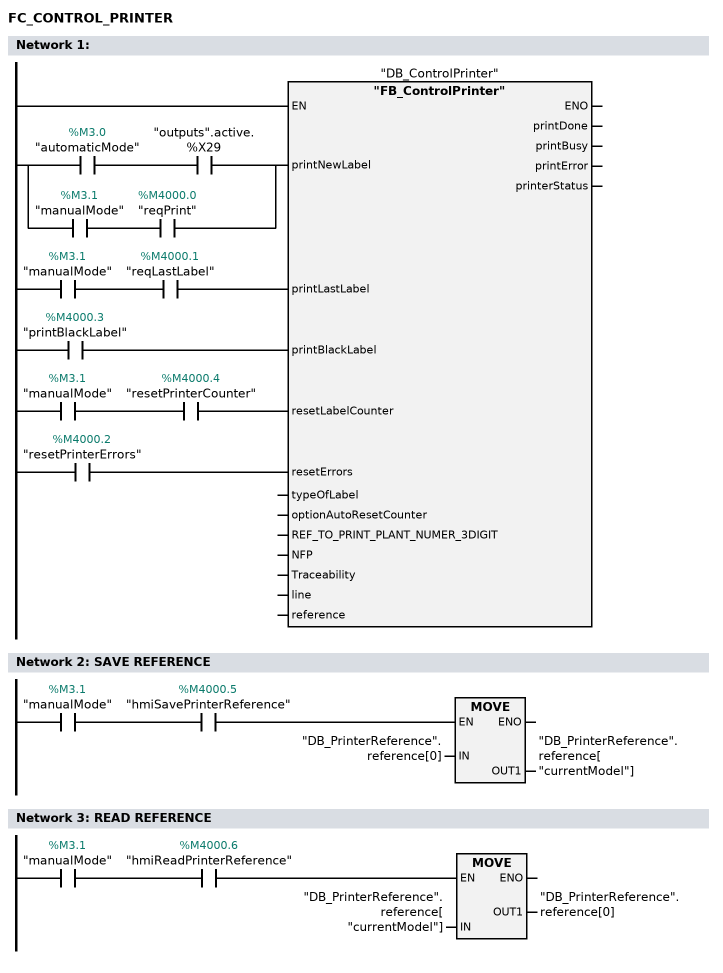
   RUNG wire#powerrail
      "DB_ControlPrinter"(printNewLabel := wire#w1, printLastLabel := wire#w2, printBlackLabel := wire#w3, resetLabelCounter := wire#w4, resetErrors := wire#w5, typeOfLabel :=, optionAutoResetCounter :=, REF_TO_PRINT_PLANT_NUMER_3DIGIT :=, NFP :=, Traceability :=, line :=, reference :=, printDone =>, printBusy =>, printError =>, printerStatus =>)
   END_RUNG
   RUNG wire#powerrail
      Contact( "automaticMode" )
      Contact( "outputs".active.%X29 )
   END_RUNG wire#w1
   RUNG wire#powerrail
      Contact( "manualMode" )
      Contact( "reqPrint" )
   END_RUNG wire#w1
   RUNG wire#powerrail
      Contact( "manualMode" )
      Contact( "reqLastLabel" )
   END_RUNG wire#w2
   RUNG wire#powerrail
      Contact( "printBlackLabel" )
   END_RUNG wire#w3
   RUNG wire#powerrail
      Contact( "manualMode" )
      Contact( "resetPrinterCounter" )
   END_RUNG wire#w4
   RUNG wire#powerrail
      Contact( "resetPrinterErrors" )
   END_RUNG wire#w5
   // the same network as SCL:
   "DB_ControlPrinter"(printNewLabel := ("automaticMode" AND "outputs".active.%X29) OR ("manualMode" AND "reqPrint"),   // "FB_ControlPrinter"
                       printLastLabel := "manualMode" AND "reqLastLabel",
                       printBlackLabel := "printBlackLabel",
                       resetLabelCounter := "manualMode" AND "resetPrinterCounter",
                       resetErrors := "resetPrinterErrors");
END_REGION

REGION Network 2: SAVE REFERENCE
   RUNG wire#powerrail
      Contact( "manualMode" )
      Contact( "hmiSavePrinterReference" )
      Move(in := "DB_PrinterReference".reference[0], out1 => "DB_PrinterReference".reference["currentModel"])
   END_RUNG
   // the same network as SCL:
   IF "manualMode" AND "hmiSavePrinterReference" THEN
       "DB_PrinterReference".reference["currentModel"] := "DB_PrinterReference".reference[0];
   END_IF;
END_REGION

REGION Network 3: READ REFERENCE
   RUNG wire#powerrail
      Contact( "manualMode" )
      Contact( "hmiReadPrinterReference" )
      Move(in := "DB_PrinterReference".reference["currentModel"], out1 => "DB_PrinterReference".reference[0])
   END_RUNG
   // the same network as SCL:
   IF "manualMode" AND "hmiReadPrinterReference" THEN
       "DB_PrinterReference".reference[0] := "DB_PrinterReference".reference["currentModel"];
   END_IF;
END_REGION
END_FUNCTION

FUNCTION_BLOCK "FB_ControlPrinter"
{ S7_Optimized_Access := 'TRUE' }
VERSION : 0.1
   VAR_INPUT 
      printNewLabel : Bool;
      printLastLabel : Bool;
      printBlackLabel : Bool;
      resetLabelCounter : Bool;
      resetErrors : Bool;
   END_VAR
   VAR_INPUT RETAIN
      typeOfLabel : Int;
   END_VAR
   VAR_INPUT 
      optionAutoResetCounter : Int;
      REF_TO_PRINT_PLANT_NUMER_3DIGIT : String[10];
      NFP : String[30];
      Traceability : Bool;
      line : String[1];
      reference : "udt_referenceMainInfo";
   END_VAR

   VAR_OUTPUT 
      printDone : Bool;
      printBusy : Bool;
      printError : Bool;
      printerStatus : Word;
   END_VAR

   VAR 
      tramToSendToPrinter : Array[0..6000] of Char;
      seqDataPreparation : Int;
      tramToPrepareToSend { S7_SetPoint := 'True'} : Array[1..20] of String;
      savePrintNewLabel : Bool;
   END_VAR
   VAR RETAIN
      "counter" : Int;
      DBcomToPrinter {InstructionName := 'TCON_IP_v4'; LibVersion := '1.0'; S7_SetPoint := 'False'} : TCON_IP_v4;
   END_VAR
   VAR 
      tSendC {InstructionName := 'TSEND_C'; LibVersion := '3.0'} : TSEND_C;
   END_VAR

   VAR_TEMP 
      dateAndTime {InstructionName := 'DTL'; LibVersion := '1.0'} : DTL;
      dateTimeStr : String;
      "date" : String[10];
      "time" : String[8];
      year : String[2];
      MFGhour : String[1];
      JulianDay : String[3];
      errCode : DInt;
      pcars : DInt;
      forCounter : Int;
      counterStr : String[4];
      cnt : DInt;
      i : Int;
      dummy : Int;
      holder : String;
      nfpToPrint : String[8];
      PN : String[8];
   END_VAR

   VAR CONSTANT 
      fieldSeparator : String := '^FS';
      RS : String := '\1E';
      GS : String := '\1D';
      EOT : String := '\04';
   END_VAR


BEGIN
	
	//***********************************************************CALCULATE DAY NUMBER **************************************
	#errCode:= RD_LOC_T(#dateAndTime);
	#dateTimeStr := "GetStrDateTime"("date" := #dateAndTime, separator := '/');
	#date := LEFT_STRING(IN := #dateTimeStr, L := 10);
	#year := MID(IN := #dateTimeStr, L := 2, P := 9);
	#time := MID(IN := #dateTimeStr, L := 8, P := 12);
	#JulianDay := "GetStrJDay"();
	#MFGhour := USINT_TO_CHAR(#dateAndTime.HOUR + 65);
	
	//********************************************* SEQUENCE MANAGE TO DATA PRINT **************************************
	//
	//>>>>>> STEP-0- >>>>>> waiting for start printing
	IF (#printNewLabel AND #seqDataPreparation = 0) THEN
	    IF #printNewLabel THEN
	        #savePrintNewLabel := TRUE;
	        #seqDataPreparation := 1;
	    END_IF;
	END_IF;
	
	//>>>>>> STEP-1- >>>>>> INITIALISE DATA TO PRINT
	IF #seqDataPreparation = 1 THEN
	    // INITILISE DATA OF TRAM TO SEND
	    // 
	    IF #typeOfLabel = 0 THEN //NO LABEL
	        FOR #i := 1 TO 20 DO
	            #tramToPrepareToSend[#i] := '';
	        END_FOR;
	        
	    ELSIF #typeOfLabel = 1 THEN //NFP LABEL
	        #tramToPrepareToSend[1] := '^XA^PW378'; //START FORMAT   
	        #tramToPrepareToSend[2] := '^BY126,126^FT169,175^BXN,7,200,0,0,1,~^FH\^FD';//DATAMATRIX
	        #tramToPrepareToSend[3] := '1234567891234567891234567891'; 
	        #tramToPrepareToSend[4] := '^FS^FT25,162^A0N,29,28^FH\^FD'; //REFERENCE
	        #tramToPrepareToSend[5] := '12345678'; 
	        #tramToPrepareToSend[6] := '^FS^FT25,124^A0N,25,24^FH\^FD'; //DATE
	        #tramToPrepareToSend[7] := 'DD/MM/YY'; //
	        #tramToPrepareToSend[8] := '^FS^FT25,87^A0N,29,28^FH\^FD'; // TIME
	        #tramToPrepareToSend[9] := 'hh:mm:ss';
	        #tramToPrepareToSend[10] := '^FS^FT26,44^A0N,29,28^FH\^FD';//DESCRIPTION
	        #tramToPrepareToSend[11] := '1234567891';
	        #tramToPrepareToSend[12] := '^FS^FT25,196^A0N,21,21^FH\^FD';//READABLE CODE
	        #tramToPrepareToSend[13] := '1234567891234567891234567891';
	        #tramToPrepareToSend[20] := '^PQ1,0,1,Y^XZ';//END FORMAT
	        #counter += 1;
	        
	    ELSIF #typeOfLabel = 2 THEN //CUSTOMER LABEL
	        #tramToPrepareToSend[1] := '^XA'; //START FORMAT   
	        #tramToPrepareToSend[2] := '^XFE:GM_FINAL.zpl';//CALL TEMPLATE
	        #tramToPrepareToSend[3] := '^FN1^FH\^FD[)>\1E06\1DY00000000000000\1DP00000000\1D12V000000000\1DT0000000000000000\1E\04^FS'; //DATAMATRIX
	        #tramToPrepareToSend[4] := '^FN2^FD1234^FS'; //GM PART NUMBER 
	        #tramToPrepareToSend[5] := '^FN3^FD5678^FS'; //GM PART NUMBER
	        #tramToPrepareToSend[6] := '^FN4^FD12345678901234^FS'; //VPPS
	        #tramToPrepareToSend[7] := '^FN5^FD123456789^FS'; //DUNS
	        #tramToPrepareToSend[8] := '^FN6^FDLSYYDDDA2B4CDSEQ^FS'; //TRACE CODE
	        #tramToPrepareToSend[9] := '^FN7^FDdd/mm/yyyy^FS'; //DATE
	        #tramToPrepareToSend[10] := '^FN8^FDhh:mm:ss^FS'; //TIME
	        #tramToPrepareToSend[11] := '^FN9^FD12345678^FS'; //FAURECIA NUMBER
	        #tramToPrepareToSend[12] := '^FN10^FD12345678^FS'; //NFP
	        #tramToPrepareToSend[13] := '^FN11^FDLINEA 3^FS'; //LINE
	        #tramToPrepareToSend[20] := '^PQ1,0,1,Y^XZ';//END FORMAT
	        #counter += 1;
	    END_IF;
	    #seqDataPreparation := 2;
	END_IF;
	
	
	//PREPARATION OF LABEL COUNTER **************************************
	#counterStr := "LabelCounterFormat"(counts := #counter, format := 'DEC', len := 3);
	IF  #counter > 999 THEN
	    #counter := 0;
	END_IF;
	
	// AUTO RESET COUNTER PER HOUR
	IF #optionAutoResetCounter = 1 THEN
	    IF #dateAndTime.MINUTE = 0 AND #dateAndTime.SECOND <= 2 THEN
	        #counter := 0;
	    END_IF;
	END_IF;
	
	
	//----------------------------------------------------------------------------------------------------------------
	//>>>>>> STEP-2- >>>>>> MODIFY CONCERNED DATA AS DATE; TIME; REFERENCE; YEAR DAY; PRODUCT REFERENCE.
	IF #seqDataPreparation = 2 THEN
	    //DATAMATRIX
	    IF #typeOfLabel = 1 THEN //NFP LABEL
	        IF #Traceability THEN
	            #tramToPrepareToSend[3] := #NFP;
	            #tramToPrepareToSend[13] := #NFP;
	        END_IF;
	        
	        IF NOT #Traceability THEN
	            #tramToPrepareToSend[3] := #line;  //line number
	            #tramToPrepareToSend[3] := CONCAT(IN1 := #tramToPrepareToSend[3], IN2 := 'P');  //label type
	            #tramToPrepareToSend[3] := CONCAT(IN1 := #tramToPrepareToSend[3], IN2 := #counterStr);  //internal sequence number
	            #tramToPrepareToSend[3] := CONCAT(IN1 := #tramToPrepareToSend[3], IN2 := #MFGhour);
	            #tramToPrepareToSend[3] := CONCAT(IN1 := #tramToPrepareToSend[3], IN2 := #JulianDay);
	            #tramToPrepareToSend[3] := CONCAT(IN1 := #tramToPrepareToSend[3], IN2 := "model".name[0]);
	            #tramToPrepareToSend[3] := CONCAT(IN1 := #tramToPrepareToSend[3], IN2 := 'R01');
	            #tramToPrepareToSend[3] := CONCAT(IN1 := #tramToPrepareToSend[3], IN2 := #REF_TO_PRINT_PLANT_NUMER_3DIGIT);
	            #tramToPrepareToSend[3] := CONCAT(IN1 := #tramToPrepareToSend[3], IN2 := #year);
	            #tramToPrepareToSend[13] := #tramToPrepareToSend[3];
	        END_IF;
	        
	        
	        //DATE
	        #tramToPrepareToSend[7] := #date;
	        
	        //TIME
	        #tramToPrepareToSend[9] := #time;
	        
	        //REFERENCE
	        #tramToPrepareToSend[5] := "model".name[0];
	        
	        //DESCRIPTION
	        #tramToPrepareToSend[11] := "model".Description[0];
	        
	        ;
	        
	        
	    ELSIF #typeOfLabel = 2 THEN //CUSTOMER LABEL
	        
	        //GM PART NUMBER 1-2
	        #tramToPrepareToSend[4] := REPLACE(IN1 := #tramToPrepareToSend[4], IN2 := (MID(IN := #reference.customerNumber, L := 4, P := 1)), L := 4, P := FIND(IN1 := #tramToPrepareToSend[4], IN2 := '1234'));
	        #tramToPrepareToSend[5] := REPLACE(IN1 := #tramToPrepareToSend[5], IN2 := (MID(IN := #reference.customerNumber, L := 4, P := 5)), L := 4, P := FIND(IN1 := #tramToPrepareToSend[5], IN2 := '5678'));
	        
	        // VPPS
	        #tramToPrepareToSend[6] := REPLACE(IN1 := #tramToPrepareToSend[6], IN2 := #reference.vpps, L := 14, P := FIND(IN1 := #tramToPrepareToSend[6], IN2 := '12345678901234'));
	        
	        // MANUFACTURING DUNS
	        #tramToPrepareToSend[7] := REPLACE(IN1 := #tramToPrepareToSend[7], IN2 := #reference.duns, L := 9, P := FIND(IN1 := #tramToPrepareToSend[7], IN2 := '123456789'));
	        
	        // TRACE CODE GM
	        //L : LINEA MACHINE
	        #tramToPrepareToSend[8] := REPLACE(IN1 := #tramToPrepareToSend[8], IN2 := #line[1], L := 1, P := (FIND(IN1 := #tramToPrepareToSend[8], IN2 := 'L')));
	        //S : SHIFT
	        #tramToPrepareToSend[8] := REPLACE(IN1 := #tramToPrepareToSend[8], IN2 := #MFGhour, L := 1, P := (FIND(IN1 := #tramToPrepareToSend[8], IN2 := 'S')));
	        //YY : YEAR
	        #tramToPrepareToSend[8] := REPLACE(IN1 := #tramToPrepareToSend[8], IN2 := #year, L := 2, P := (FIND(IN1 := #tramToPrepareToSend[8], IN2 := 'YY')));
	        //DDD : JULIAN DAY
	        #tramToPrepareToSend[8] := REPLACE(IN1 := #tramToPrepareToSend[8], IN2 := #JulianDay, L := 3, P := (FIND(IN1 := #tramToPrepareToSend[8], IN2 := 'DDD')));
	        //REF FAS 
	        #tramToPrepareToSend[8] := REPLACE(IN1 := #tramToPrepareToSend[8], IN2 := RIGHT(IN := #reference.partNumber, L := 4), L := 4, P := (FIND(IN1 := #tramToPrepareToSend[8], IN2 := 'A2B4')));
	        //REV
	        #tramToPrepareToSend[8] := REPLACE(IN1 := #tramToPrepareToSend[8], IN2 := LEFT(IN := #reference.rev, L := 2), L := 2, P := (FIND(IN1 := #tramToPrepareToSend[8], IN2 := 'CD')));
	        //SEQN : LABEL COUNTER
	        #tramToPrepareToSend[8] := REPLACE(IN1 := #tramToPrepareToSend[8], IN2 := RIGHT(IN := #counterStr, L := 3), L := 3, P := (FIND(IN1 := #tramToPrepareToSend[8], IN2 := 'SEQ')));
	        
	        
	        //Data Matrix
	        //Y : VPPS
	        #tramToPrepareToSend[3] := REPLACE(IN1 := #tramToPrepareToSend[3], IN2 := LEFT(IN := #reference.vpps, L := 14), L := 14, P := (FIND(IN1 := #tramToPrepareToSend[3], IN2 := 'Y') + 1));
	        //P : GM PART NUMBER
	        #tramToPrepareToSend[3] := REPLACE(IN1 := #tramToPrepareToSend[3], IN2 := LEFT(IN := #reference.customerNumber, L := 8), L := 8, P := (FIND(IN1 := #tramToPrepareToSend[3], IN2 := 'P') + 1));
	        //V : DUNS
	        #tramToPrepareToSend[3] := REPLACE(IN1 := #tramToPrepareToSend[3], IN2 := LEFT(IN := #reference.duns, L := 9), L := 9, P := (FIND(IN1 := #tramToPrepareToSend[3], IN2 := 'V') + 1));
	        //T : GM TRACE CODE
	        #tramToPrepareToSend[3] := REPLACE(IN1 := #tramToPrepareToSend[3], IN2 := MID(IN := #tramToPrepareToSend[8], L := 16, P := 8), L := 16, P := (FIND(IN1 := #tramToPrepareToSend[3], IN2 := 'T') + 1));
	        //DATE
	        #tramToPrepareToSend[9] := REPLACE(IN1 := #tramToPrepareToSend[9], IN2 := #date, L := 10, P := (FIND(IN1 := #tramToPrepareToSend[9], IN2 := 'dd/mm/yyyy')));
	        //TIME
	        #tramToPrepareToSend[10] := REPLACE(IN1 := #tramToPrepareToSend[10], IN2 := #time, L := 8, P := (FIND(IN1 := #tramToPrepareToSend[10], IN2 := 'hh:mm:ss')));
	        //FAURECIA NUMBER
	        #PN := MID(IN := #NFP, L := 8, P := 9);
	        #tramToPrepareToSend[11] := REPLACE(IN1 := #tramToPrepareToSend[11], IN2 := #PN, L := 8, P := (FIND(IN1 := #tramToPrepareToSend[11], IN2 := '12345678')));
	        //NFP
	        #nfpToPrint := LEFT(IN := #NFP, L := 8);
	        #tramToPrepareToSend[12] := REPLACE(IN1 := #tramToPrepareToSend[12], IN2 := #nfpToPrint, L := 8, P := (FIND(IN1 := #tramToPrepareToSend[12], IN2 := '12345678')));
	    END_IF;
	    #seqDataPreparation := 3;
	END_IF;
	
	
	//>>>>>> STEP-3- >>>>>> COPY TO TRAM PRINTER TO SEND
	IF #seqDataPreparation = 3 THEN
	    //RESET DB TRAM TO SEND 
	    FILL_BLK(IN := ' ',
	             COUNT := 6000,
	             OUT => #tramToSendToPrinter[0]);
	    #pcars := 0;
	   // FILL TRAM TO SEND TO PRINTER
	    FOR #forCounter := 1 TO 20 DO
	        Strg_TO_Chars(Strg := #tramToPrepareToSend[#forCounter],
	                      pChars := #pcars,
	                      Cnt => #cnt,
	                      Chars := #tramToSendToPrinter);
	        #pcars := #pcars + #cnt;
	    END_FOR;
	    #seqDataPreparation := 4;
	END_IF;
	
	// CONNECTION TO PRINTER PARAMETERS
	#DBcomToPrinter.ConnectionType := 16#0B;
	#DBcomToPrinter.InterfaceId := 64;
	#DBcomToPrinter.ID := 10;
	#DBcomToPrinter.ActiveEstablished := TRUE;
	#DBcomToPrinter.LocalPort := 0;
	#tSendC(REQ:=(#seqDataPreparation = 4),
	        CONT:=TRUE,
	        LEN:=0,
	        DONE=>#printDone,
	        BUSY=>#printBusy,
	        ERROR=>#printError,
	        STATUS=>#printerStatus,
	        CONNECT:=#DBcomToPrinter,
	        DATA:=#tramToSendToPrinter
	);
	IF #seqDataPreparation = 4 AND #printNewLabel THEN
	    #printDone := TRUE;
	    ;
	END_IF;
	
	
	//>>>>>> STEP-X- >>>>>> END OF SEQUENCE: WAITING 
	//
	IF #seqDataPreparation = 4 AND NOT (#printNewLabel) THEN
	    #printDone := FALSE;
	    #savePrintNewLabel := FALSE;
	    #seqDataPreparation := 0;
	END_IF;
	
	
END_FUNCTION_BLOCK

FUNCTION "GetStrJDay" : String
{ S7_Optimized_Access := 'TRUE' }
VERSION : 0.1
   VAR_TEMP 
      julianDayDint : DInt;
      DateTime {InstructionName := 'DTL'; LibVersion := '1.0'} : DTL;
      return : Int;
      LeapYear : DInt;
      julianDayHolder : String;
   END_VAR

   VAR CONSTANT 
      "__JAN" : USInt := 1;
      "__FEB" : USInt := 2;
      "__MAR" : USInt := 3;
      "__APR" : USInt := 4;
      "__MAY" : USInt := 5;
      "__JUN" : USInt := 6;
      "__JUL" : USInt := 7;
      "__AUG" : USInt := 8;
      "__SEP" : USInt := 9;
      "__OCT" : USInt := 10;
      "__NOV" : USInt := 11;
      "__DEC" : USInt := 12;
   END_VAR


BEGIN
	#return := RD_LOC_T(#DateTime);
	#LeapYear := #DateTime.YEAR MOD 4;
	
	//CALC JDAY
	CASE #DateTime.MONTH OF
	    #"__JAN": #julianDayDint := #DateTime.DAY;
	    #"__FEB": #julianDayDint := (#DateTime.DAY + DINT#31);
	    #"__MAR": #julianDayDint := (#DateTime.DAY + DINT#59);
	    #"__APR": #julianDayDint := (#DateTime.DAY + DINT#90);
	    #"__MAY": #julianDayDint := (#DateTime.DAY + DINT#120);
	    #"__JUN": #julianDayDint := (#DateTime.DAY + DINT#151);
	    #"__JUL": #julianDayDint := (#DateTime.DAY + DINT#181);
	    #"__AUG": #julianDayDint := (#DateTime.DAY + DINT#212);
	    #"__SEP": #julianDayDint := (#DateTime.DAY + DINT#243);
	    #"__OCT": #julianDayDint := (#DateTime.DAY + DINT#273);
	    #"__NOV": #julianDayDint := (#DateTime.DAY + DINT#304);
	    #"__DEC": #julianDayDint := (#DateTime.DAY + DINT#334);
	END_CASE;
	
	//IF LEAP YEAR
	IF #LeapYear = 0 AND #DateTime.MONTH > 2 THEN
	    #julianDayDint := #julianDayDint + 1;
	    ;
	END_IF;
	
	//JULIAN DAY IN STRING FORMAT
	#julianDayHolder := DINT_TO_STRING(IN := ABS_DINT(IN := #julianDayDint));
	#julianDayHolder := DELETE(IN := #julianDayHolder, L := 1, P := 1);
	IF #julianDayDint < 10 THEN
	    #GetStrJDay := CONCAT_STRING(IN1 := '00', IN2 := #julianDayHolder);
	ELSIF #julianDayDint >= 10 AND #julianDayDint < 100 THEN
	    #GetStrJDay := CONCAT_STRING(IN1 := '0', IN2 := #julianDayHolder);
	ELSE
	    #GetStrJDay := #julianDayHolder;
	END_IF;
	
	
END_FUNCTION

FUNCTION "LabelCounterFormat" : String
{ S7_Optimized_Access := 'TRUE' }
VERSION : 0.1
   VAR_INPUT 
      counts : Int;
      format : String;
      len : Int;
   END_VAR

   VAR_TEMP 
      tempCounter : String;
      i : Int;
      errCode : Word;
   END_VAR


BEGIN
	
	IF #format = 'DEC' THEN
	    VAL_STRG(IN := #counts,
	             SIZE := INT_TO_USINT( #len),
	             PREC := 0,
	             FORMAT := 0,
	             P := 1,
	             OUT => #tempCounter);
	    FOR #i := 0 TO #len DO
	        IF (FIND(IN1 := #tempCounter, IN2 := ' ') > 0) THEN
	            #tempCounter := REPLACE(IN1 := #tempCounter, IN2 := '0', L := 1, P := FIND(IN1 := #tempCounter, IN2 := ' '));
	        END_IF;
	    END_FOR;
	ELSIF #format = 'HEX' THEN
	    #errCode := HTA(IN := #counts, N := INT_TO_USINT(#len), OUT => #tempCounter);
	
	END_IF;
	#LabelCounterFormat := #tempCounter;
END_FUNCTION

FUNCTION_BLOCK "FC_IJCORE_MAIN"   // FB1000, LAD
{ S7_Optimized_Access := 'FALSE' }
VERSION : 0.1
// stored: AutoNumber false, IsIECCheckEnabled false, SetENOAutomatically false, UDAEnableTagReadback false
   VAR DB_SPECIFIC
      Enable : Bool;
      Mode : Int;
      Indicator : Int;
      AlarmReset : Bool;
      NFP : Array[1..5] of String[30];
   END_VAR
   VAR
      AWK : "FB_IJC_AWAKE_SIGNAL";
      MSG : Array[1..20] of "FB_IJC_PROTOCOL";
   END_VAR
   VAR DB_SPECIFIC
      Faults : Array[0..1] of Word;
   END_VAR
   VAR
      FaultsArray AT Faults : Array[1..32] of Bool;
   END_VAR
   VAR_TEMP
      "return" : Bool;
      i : Int;
      ERROR_STR : String;
   END_VAR
BEGIN

REGION Network 1: Fault Reset
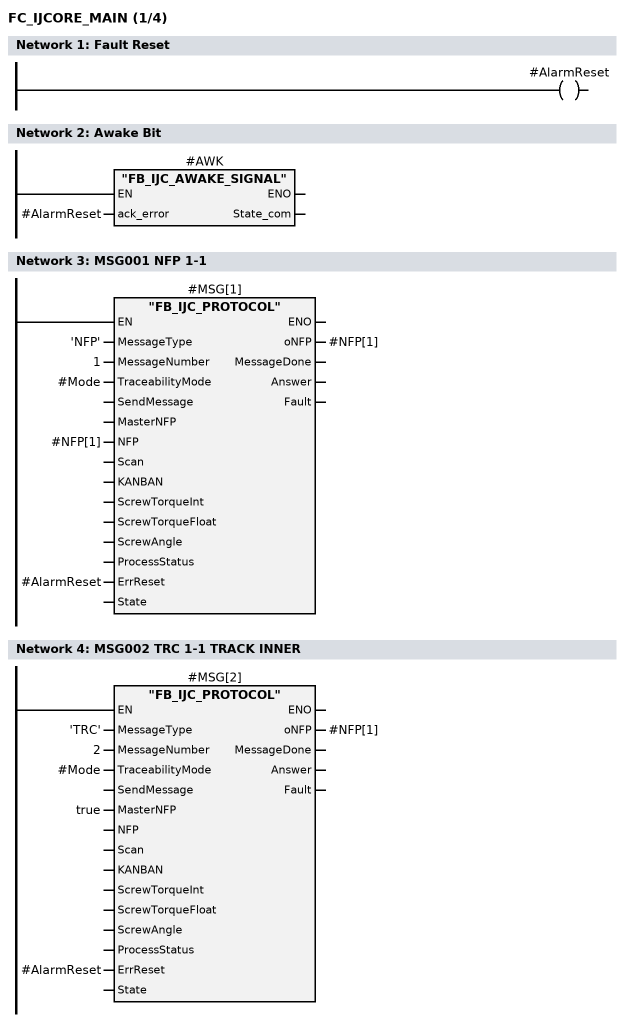
   RUNG wire#powerrail
      Coil( #AlarmReset )
   END_RUNG
   // the same network as SCL:
   #AlarmReset := TRUE;
END_REGION

REGION Network 2: Awake Bit
   RUNG wire#powerrail
      #AWK(ack_error := #AlarmReset, State_com =>)
   END_RUNG
   // the same network as SCL:
   #AWK(ack_error := #AlarmReset);   // "FB_IJC_AWAKE_SIGNAL"
END_REGION

REGION Network 3: MSG001 NFP 1-1
   RUNG wire#powerrail
      #MSG[1](MessageType := 'NFP', MessageNumber := 1, TraceabilityMode := #Mode, SendMessage :=, MasterNFP :=, NFP := #NFP[1], Scan :=, KANBAN :=, ScrewTorqueInt :=, ScrewTorqueFloat :=, ScrewAngle :=, ProcessStatus :=, ErrReset := #AlarmReset, State :=, oNFP => #NFP[1], MessageDone =>, Answer =>, Fault =>)
   END_RUNG
   // the same network as SCL:
   #MSG[1](MessageType := 'NFP',   // "FB_IJC_PROTOCOL"
           MessageNumber := 1,
           TraceabilityMode := #Mode,
           NFP := #NFP[1],
           ErrReset := #AlarmReset,
           oNFP => #NFP[1]);
END_REGION

REGION Network 4: MSG002 TRC 1-1 TRACK INNER
   RUNG wire#powerrail
      #MSG[2](MessageType := 'TRC', MessageNumber := 2, TraceabilityMode := #Mode, SendMessage :=, MasterNFP := true, NFP :=, Scan :=, KANBAN :=, ScrewTorqueInt :=, ScrewTorqueFloat :=, ScrewAngle :=, ProcessStatus :=, ErrReset := #AlarmReset, State :=, oNFP => #NFP[1], MessageDone =>, Answer =>, Fault =>)
   END_RUNG
   // the same network as SCL:
   #MSG[2](MessageType := 'TRC',   // "FB_IJC_PROTOCOL"
           MessageNumber := 2,
           TraceabilityMode := #Mode,
           MasterNFP := true,
           ErrReset := #AlarmReset,
           oNFP => #NFP[1]);
END_REGION

REGION Network 5: MSG003 TRC 1-2 TRACK OUTER
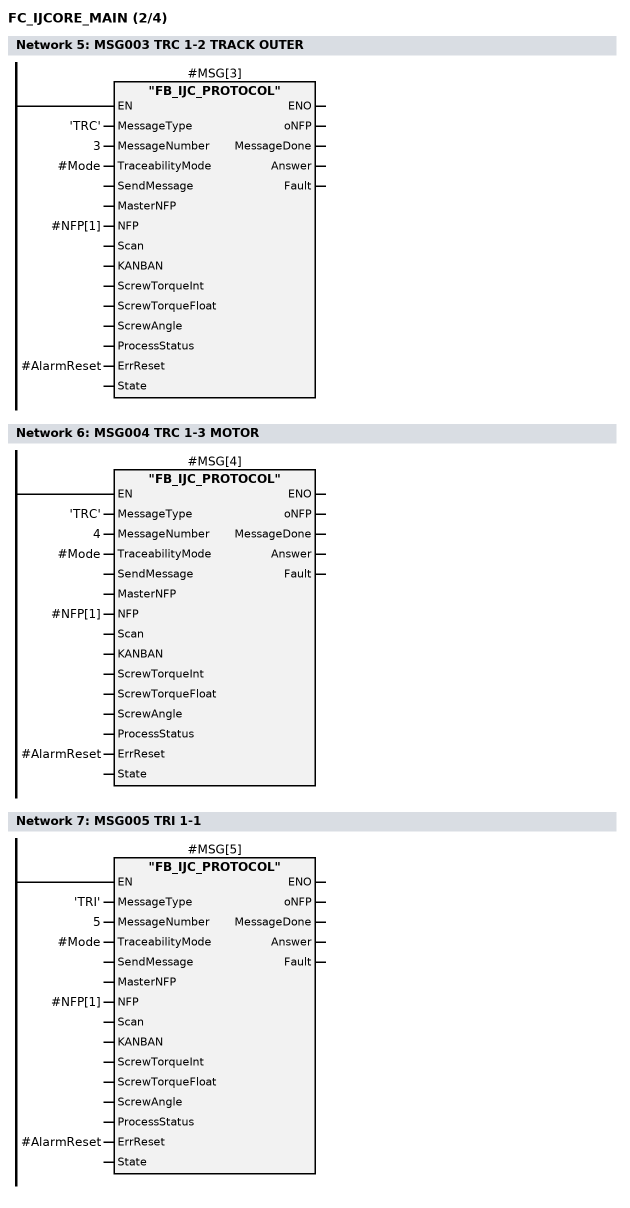
   RUNG wire#powerrail
      #MSG[3](MessageType := 'TRC', MessageNumber := 3, TraceabilityMode := #Mode, SendMessage :=, MasterNFP :=, NFP := #NFP[1], Scan :=, KANBAN :=, ScrewTorqueInt :=, ScrewTorqueFloat :=, ScrewAngle :=, ProcessStatus :=, ErrReset := #AlarmReset, State :=, oNFP =>, MessageDone =>, Answer =>, Fault =>)
   END_RUNG
   // the same network as SCL:
   #MSG[3](MessageType := 'TRC',   // "FB_IJC_PROTOCOL"
           MessageNumber := 3,
           TraceabilityMode := #Mode,
           NFP := #NFP[1],
           ErrReset := #AlarmReset);
END_REGION

REGION Network 6: MSG004 TRC 1-3 MOTOR
   RUNG wire#powerrail
      #MSG[4](MessageType := 'TRC', MessageNumber := 4, TraceabilityMode := #Mode, SendMessage :=, MasterNFP :=, NFP := #NFP[1], Scan :=, KANBAN :=, ScrewTorqueInt :=, ScrewTorqueFloat :=, ScrewAngle :=, ProcessStatus :=, ErrReset := #AlarmReset, State :=, oNFP =>, MessageDone =>, Answer =>, Fault =>)
   END_RUNG
   // the same network as SCL:
   #MSG[4](MessageType := 'TRC',   // "FB_IJC_PROTOCOL"
           MessageNumber := 4,
           TraceabilityMode := #Mode,
           NFP := #NFP[1],
           ErrReset := #AlarmReset);
END_REGION

REGION Network 7: MSG005 TRI 1-1
   RUNG wire#powerrail
      #MSG[5](MessageType := 'TRI', MessageNumber := 5, TraceabilityMode := #Mode, SendMessage :=, MasterNFP :=, NFP := #NFP[1], Scan :=, KANBAN :=, ScrewTorqueInt :=, ScrewTorqueFloat :=, ScrewAngle :=, ProcessStatus :=, ErrReset := #AlarmReset, State :=, oNFP =>, MessageDone =>, Answer =>, Fault =>)
   END_RUNG
   // the same network as SCL:
   #MSG[5](MessageType := 'TRI',   // "FB_IJC_PROTOCOL"
           MessageNumber := 5,
           TraceabilityMode := #Mode,
           NFP := #NFP[1],
           ErrReset := #AlarmReset);
END_REGION

REGION Network 8: MSG006 CNF 1-1 TRACK INNER
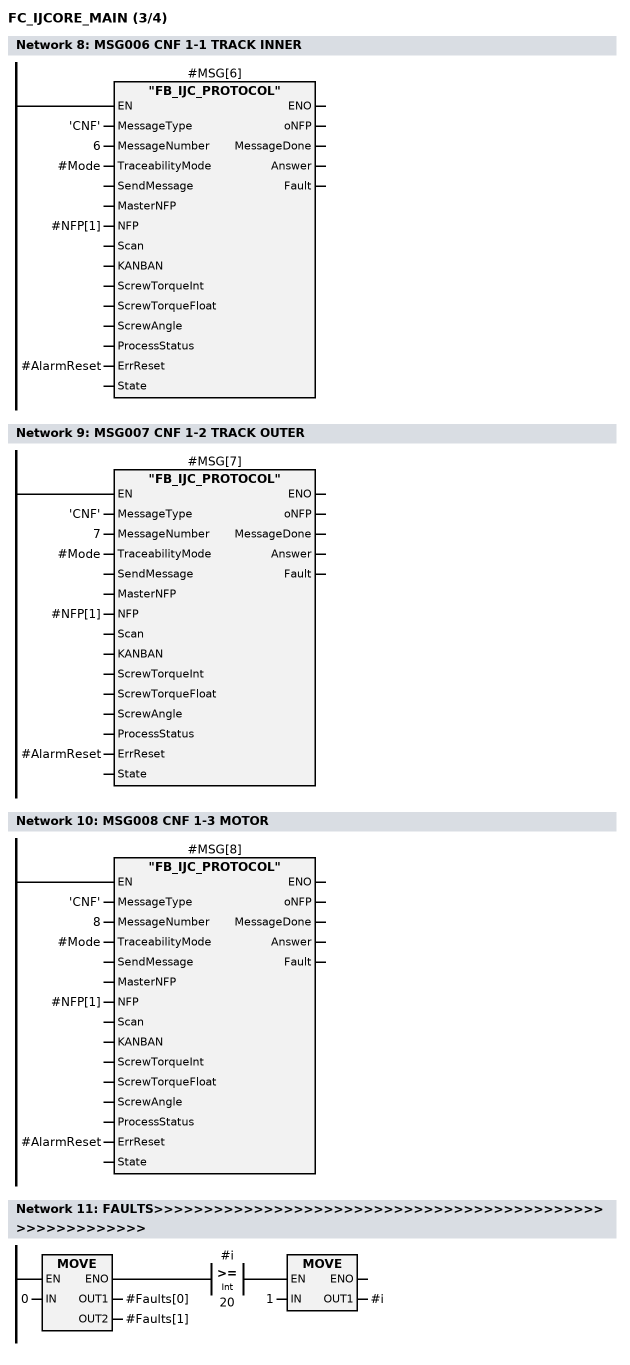
   RUNG wire#powerrail
      #MSG[6](MessageType := 'CNF', MessageNumber := 6, TraceabilityMode := #Mode, SendMessage :=, MasterNFP :=, NFP := #NFP[1], Scan :=, KANBAN :=, ScrewTorqueInt :=, ScrewTorqueFloat :=, ScrewAngle :=, ProcessStatus :=, ErrReset := #AlarmReset, State :=, oNFP =>, MessageDone =>, Answer =>, Fault =>)
   END_RUNG
   // the same network as SCL:
   #MSG[6](MessageType := 'CNF',   // "FB_IJC_PROTOCOL"
           MessageNumber := 6,
           TraceabilityMode := #Mode,
           NFP := #NFP[1],
           ErrReset := #AlarmReset);
END_REGION

REGION Network 9: MSG007 CNF 1-2 TRACK OUTER
   RUNG wire#powerrail
      #MSG[7](MessageType := 'CNF', MessageNumber := 7, TraceabilityMode := #Mode, SendMessage :=, MasterNFP :=, NFP := #NFP[1], Scan :=, KANBAN :=, ScrewTorqueInt :=, ScrewTorqueFloat :=, ScrewAngle :=, ProcessStatus :=, ErrReset := #AlarmReset, State :=, oNFP =>, MessageDone =>, Answer =>, Fault =>)
   END_RUNG
   // the same network as SCL:
   #MSG[7](MessageType := 'CNF',   // "FB_IJC_PROTOCOL"
           MessageNumber := 7,
           TraceabilityMode := #Mode,
           NFP := #NFP[1],
           ErrReset := #AlarmReset);
END_REGION

REGION Network 10: MSG008 CNF 1-3 MOTOR
   RUNG wire#powerrail
      #MSG[8](MessageType := 'CNF', MessageNumber := 8, TraceabilityMode := #Mode, SendMessage :=, MasterNFP :=, NFP := #NFP[1], Scan :=, KANBAN :=, ScrewTorqueInt :=, ScrewTorqueFloat :=, ScrewAngle :=, ProcessStatus :=, ErrReset := #AlarmReset, State :=, oNFP =>, MessageDone =>, Answer =>, Fault =>)
   END_RUNG
   // the same network as SCL:
   #MSG[8](MessageType := 'CNF',   // "FB_IJC_PROTOCOL"
           MessageNumber := 8,
           TraceabilityMode := #Mode,
           NFP := #NFP[1],
           ErrReset := #AlarmReset);
END_REGION

REGION Network 11: FAULTS>>>>>>>>>>>>>>>>>>>>>>>>>>>>>>>>>>>>>>>>>>>>>>>>>>>>>>>>>>
   RUNG wire#powerrail
      Move(in := 0, out1 => #Faults[0], out2 => #Faults[1])
      { S7_Templates := "SrcType := Int" } GE_Contact(in1 := #i, in2 := 20)
      Move(in := 1, out1 => #i)
   END_RUNG
   // the same network as SCL:
   #Faults[0] := 0;
   #Faults[1] := 0;
   IF #i >= 20 THEN #i := 1; END_IF;
END_REGION

REGION Network 12: Awake bit
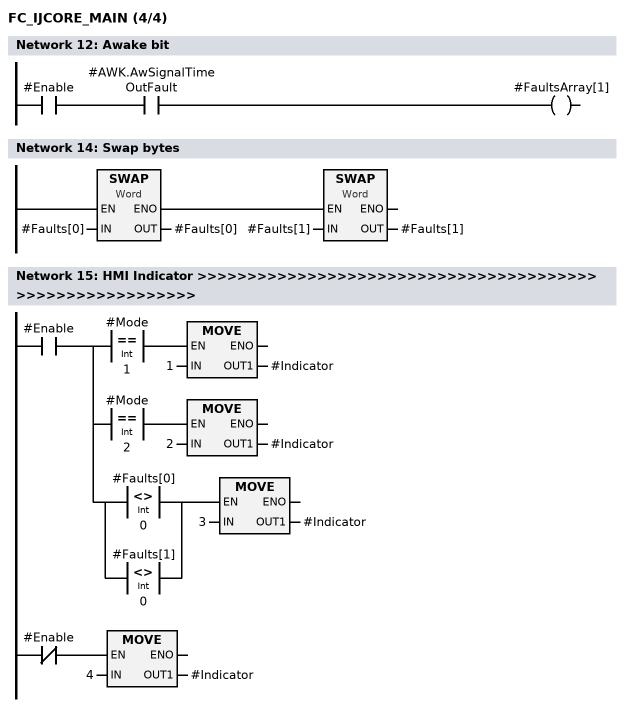
   RUNG wire#powerrail
      Contact( #Enable )
      Contact( #AWK.AwSignalTimeOutFault )
      Coil( #FaultsArray[1] )
   END_RUNG
   // the same network as SCL:
   #FaultsArray[1] := #Enable AND #AWK.AwSignalTimeOutFault;
END_REGION

REGION Network 13 (SCL): Answer faults
   FOR #i := 1 TO 20 DO
       CASE #MSG[#i].Answer OF
           -2:  // NFP not founded
               #FaultsArray[2] := TRUE;
           -3:  //Part number NOT inside BOM
               #FaultsArray[3] := TRUE;
           -4: // PFC not ok
               #FaultsArray[4] := TRUE;
           -5: //Component already used
               #FaultsArray[5] := true;
           -6: //Module already used
               #FaultsArray[6] := true;
           -10: //Status NOK from previous operation
               #FaultsArray[10] := true;

       END_CASE;



   END_FOR;
END_REGION

REGION Network 14: Swap bytes
   #Faults[0] := SWAP(#Faults[0]);
   #Faults[1] := SWAP(#Faults[1]);
END_REGION

REGION Network 15: HMI Indicator >>>>>>>>>>>>>>>>>>>>>>>>>>>>>>>>>>>>>>>>>>>>>>>>>>>>>>>>>>
   RUNG wire#powerrail
      Contact( #Enable )
      wire#w1
      { S7_Templates := "SrcType := Int" } EQ_Contact(in1 := #Mode, in2 := 1)
      Move(in := 1, out1 => #Indicator)
   END_RUNG
   RUNG wire#w1
      { S7_Templates := "SrcType := Int" } EQ_Contact(in1 := #Mode, in2 := 2)
      Move(in := 2, out1 => #Indicator)
   END_RUNG
   RUNG wire#w1
      { S7_Templates := "SrcType := Int" } NE_Contact(in1 := #Faults[0], in2 := 0)
      wire#w2
      Move(in := 3, out1 => #Indicator)
   END_RUNG
   RUNG wire#w1
      { S7_Templates := "SrcType := Int" } NE_Contact(in1 := #Faults[1], in2 := 0)
   END_RUNG wire#w2
   RUNG wire#powerrail
      I_Contact( #Enable )
      Move(in := 4, out1 => #Indicator)
   END_RUNG
   // the same network as SCL:
   IF #Enable AND (#Mode = 1) THEN #Indicator := 1; END_IF;
   IF #Enable AND (#Mode = 2) THEN #Indicator := 2; END_IF;
   IF #Enable AND ((#Faults[0] <> 0) OR (#Faults[1] <> 0)) THEN #Indicator := 3; END_IF;
   IF NOT #Enable THEN #Indicator := 4; END_IF;
END_REGION
END_FUNCTION_BLOCK

FUNCTION_BLOCK "FB_IJC_AWAKE_SIGNAL"   // FB1003, LAD
TITLE = Awake signal
{ S7_Optimized_Access := 'TRUE' }
VERSION : 0.1
// This function supervise Awake signal, 
// - Awake signal is to test communication between PLC and IJCORE. 
// - Awake signal is set to 1 by PLC and set to -1 by IJCORE alternatively.
// - first PLC check if awake signal is different of 1, if it is, PLC launch timer T1 
//  (1s<T1<10s). at the end of this temporisation, PLC set awake signal to 1 and 
//  launch Timer 2. 
// - if IJCORE don't set awake signal to -1 before the end of timer 2,PLC generate  
//   Time out fault for awake signal.
// stored: AutoNumber false, IsIECCheckEnabled false, IsRetainMemResEnabled false, MemoryReserve 100, SetENOAutomatically false, UDAEnableTagReadback false
   VAR_INPUT
      ack_error : Bool;
   END_VAR
   VAR_OUTPUT
      State_com : SInt;
   END_VAR
   VAR
      T1PresetValue : Time := T#1S;
      T2PresetValue : Time := T#60S;
      AwSignalTimeOutFault : Bool := 0;
      Reset_Counters : Bool;
      Restart_Counter_bit_of_life : USInt := 0;
      NB_Bit_of_Life : Bool;
      number_restart : DInt;
      check_restart : Bool;
      "Timer" { ExternalAccessible := 'False'; ExternalVisible := 'False'; ExternalWritable := 'False'} : Array[1..5] of TON_TIME;
   END_VAR
   VAR CONSTANT
      Trestart : Time := T#200ms;
      T3 : Time := T#2s;
   END_VAR
   VAR_TEMP   // added for the SCL form of the ladder/FBD networks
      _w1 : Bool;
   END_VAR
BEGIN

REGION Network 1: - if awake signal is -1 then launch timer 1
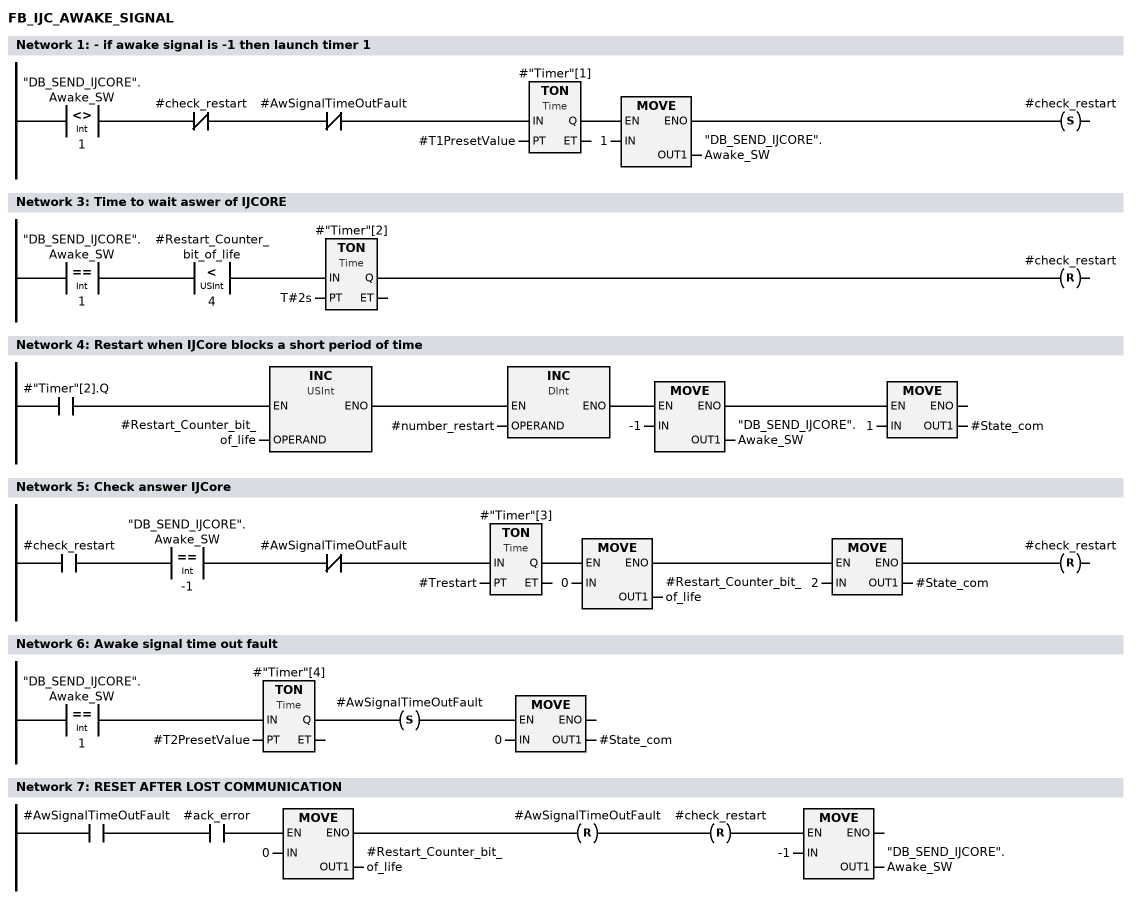
   RUNG wire#powerrail
      { S7_Templates := "SrcType := Int" } NE_Contact(in1 := "DB_SEND_IJCORE".Awake_SW, in2 := 1)
      I_Contact( #check_restart )
      I_Contact( #AwSignalTimeOutFault )
      { S7_Templates := "time_type := Time" } #"Timer"[1].TON(pt := #T1PresetValue, et =>)
      Move(in := 1, out1 => "DB_SEND_IJCORE".Awake_SW)
      S_Coil( #check_restart )
   END_RUNG
   // the same network as SCL:
   #"Timer"[1].TON(IN := ("DB_SEND_IJCORE".Awake_SW <> 1) AND NOT #check_restart AND NOT #AwSignalTimeOutFault,
                   PT := #T1PresetValue);
   IF #"Timer"[1].Q THEN
       "DB_SEND_IJCORE".Awake_SW := 1;
       #check_restart := TRUE;
   END_IF;
END_REGION

REGION Network 2: Diagnostic
END_REGION

REGION Network 3: Time to wait aswer of IJCORE
   RUNG wire#powerrail
      { S7_Templates := "SrcType := Int" } EQ_Contact(in1 := "DB_SEND_IJCORE".Awake_SW, in2 := 1)
      { S7_Templates := "SrcType := USInt" } LT_Contact(in1 := #Restart_Counter_bit_of_life, in2 := 4)
      { S7_Templates := "time_type := Time" } #"Timer"[2].TON(pt := T#2s, et =>)
      R_Coil( #check_restart )
   END_RUNG
   // the same network as SCL:
   #"Timer"[2].TON(IN := ("DB_SEND_IJCORE".Awake_SW = 1) AND (#Restart_Counter_bit_of_life < 4), PT := T#2s);
   IF #"Timer"[2].Q THEN #check_restart := FALSE; END_IF;
END_REGION

REGION Network 4: Restart when IJCore blocks a short period of time
   RUNG wire#powerrail
      Contact( #"Timer"[2].Q )
      { S7_Templates := "DestType := USInt" } Inc( #Restart_Counter_bit_of_life )
      { S7_Templates := "DestType := DInt" } Inc( #number_restart )
      Move(in := -1, out1 => "DB_SEND_IJCORE".Awake_SW)
      Move(in := 1, out1 => #State_com)
   END_RUNG
   // the same network as SCL:
   IF #"Timer"[2].Q THEN
       #Restart_Counter_bit_of_life := #Restart_Counter_bit_of_life + 1;
       #number_restart := #number_restart + 1;
       "DB_SEND_IJCORE".Awake_SW := -1;
       #State_com := 1;
   END_IF;
END_REGION

REGION Network 5: Check answer IJCore
   RUNG wire#powerrail
      Contact( #check_restart )
      { S7_Templates := "SrcType := Int" } EQ_Contact(in1 := "DB_SEND_IJCORE".Awake_SW, in2 := -1)
      I_Contact( #AwSignalTimeOutFault )
      { S7_Templates := "time_type := Time" } #"Timer"[3].TON(pt := #Trestart, et =>)
      Move(in := 0, out1 => #Restart_Counter_bit_of_life)
      Move(in := 2, out1 => #State_com)
      R_Coil( #check_restart )
   END_RUNG
   // the same network as SCL:
   #"Timer"[3].TON(IN := #check_restart AND ("DB_SEND_IJCORE".Awake_SW = (-1)) AND NOT #AwSignalTimeOutFault,
                   PT := #Trestart);
   IF #"Timer"[3].Q THEN
       #Restart_Counter_bit_of_life := 0;
       #State_com := 2;
       #check_restart := FALSE;
   END_IF;
END_REGION

REGION Network 6: Awake signal time out fault
   RUNG wire#powerrail
      { S7_Templates := "SrcType := Int" } EQ_Contact(in1 := "DB_SEND_IJCORE".Awake_SW, in2 := 1)
      { S7_Templates := "time_type := Time" } #"Timer"[4].TON(pt := #T2PresetValue, et =>)
      S_Coil( #AwSignalTimeOutFault )
      Move(in := 0, out1 => #State_com)
   END_RUNG
   // the same network as SCL:
   #"Timer"[4].TON(IN := "DB_SEND_IJCORE".Awake_SW = 1, PT := #T2PresetValue);
   IF #"Timer"[4].Q THEN
       #AwSignalTimeOutFault := TRUE;
       #State_com := 0;
   END_IF;
END_REGION

REGION Network 7: RESET AFTER LOST COMMUNICATION
   RUNG wire#powerrail
      Contact( #AwSignalTimeOutFault )
      Contact( #ack_error )
      Move(in := 0, out1 => #Restart_Counter_bit_of_life)
      R_Coil( #AwSignalTimeOutFault )
      R_Coil( #check_restart )
      Move(in := -1, out1 => "DB_SEND_IJCORE".Awake_SW)
   END_RUNG
   // the same network as SCL:
   IF #AwSignalTimeOutFault AND #ack_error THEN #Restart_Counter_bit_of_life := 0; END_IF;
   #_w1 := #AwSignalTimeOutFault AND #ack_error;
   IF #_w1 THEN
       #AwSignalTimeOutFault := FALSE;
       #check_restart := FALSE;
       "DB_SEND_IJCORE".Awake_SW := -1;
   END_IF;
END_REGION
END_FUNCTION_BLOCK

FUNCTION_BLOCK "FB_IJC_PROTOCOL"
TITLE = IJCORE PROTOCOL
{ S7_Optimized_Access := 'TRUE' }
AUTHOR : 'R.ROBINS'
VERSION : 0.1
   VAR_INPUT 
      MessageType : String[3];
      MessageNumber { ExternalVisible := 'False'; ExternalWritable := 'False'} : DInt;
      TraceabilityMode : Int;
      SendMessage { ExternalVisible := 'False'; ExternalWritable := 'False'} : Bool;
      MasterNFP : Bool;
      NFP : String[30];
      Scan : String[80];
      KANBAN : String[11];
      ScrewTorqueInt : Word;
      ScrewTorqueFloat : Word;
      ScrewAngle : Word;
      ProcessStatus { ExternalAccessible := 'False'; ExternalVisible := 'False'; ExternalWritable := 'False'} : USInt;
      ErrReset { ExternalAccessible := 'False'; ExternalVisible := 'False'; ExternalWritable := 'False'} : Bool;
   END_VAR

   VAR_OUTPUT 
      oNFP : String[30];
      MessageDone : Bool;
      Answer : Int;
      Fault : DInt;
   END_VAR

   VAR_IN_OUT 
      State { ExternalAccessible := 'False'; ExternalVisible := 'False'; ExternalWritable := 'False'} : Int;
   END_VAR

   VAR 
      SEND_OFFSET { ExternalAccessible := 'False'; ExternalVisible := 'False'; ExternalWritable := 'False'} : Struct
         SW { ExternalAccessible := 'False'; ExternalVisible := 'False'; ExternalWritable := 'False'} : DInt;
         MSG { ExternalAccessible := 'False'; ExternalVisible := 'False'; ExternalWritable := 'False'} : DInt;
      END_STRUCT;
      REC_OFFSET { ExternalAccessible := 'False'; ExternalVisible := 'False'; ExternalWritable := 'False'} : Struct
         SW { ExternalAccessible := 'False'; ExternalVisible := 'False'; ExternalWritable := 'False'} : DInt;
         MSG { ExternalAccessible := 'False'; ExternalVisible := 'False'; ExternalWritable := 'False'} : DInt;
         ANS { ExternalAccessible := 'False'; ExternalVisible := 'False'; ExternalWritable := 'False'} : DInt;
      END_STRUCT;
      ONS : Array[1..8] of Bool;
   END_VAR

   VAR_TEMP 
      IDB : Int;
      i : Int;
      j : Int;
      k : Int;
      CNT : Int;
      CNT_STR : String[2];
      MSG : DInt;
      ErrCode : Int;
   END_VAR

   VAR CONSTANT 
      "DB" : Byte := 16#84;
      CLEAR : Word := 16#0000;
      MINUS1 : Word := 16#FFFF;
      PLUS1 : Word := 16#0001;
      DB_REC : DB_ANY := 1006;
      DB_SEND : DB_ANY := 1005;
      "_CNF_" : Int := 1;
      "_TRS_" : Int := 2;
      "_TRI_" : Int := 3;
      "_TRE_" : Int := 4;
      "_STA_" : Int := 5;
      "_ANDON_" : Int := 6;
      "_TRR_" : Int := 7;
      "_TRW_" : Int := 8;
      "_PFC_" : Int := 9;
      "_NFP_" : Int := 10;
      "_CMA_" : Int := 11;
      "_TMA_" : Int := 12;
      "_TRB_" : Int := 13;
      Blank : String := '';
   END_VAR


BEGIN
	//TITLE = 'IJCORE PROTOCOL'
	//AUTHOR: RAUL ROBINS
	//CREATED ON: 03/24/2023
	//VERSION: 3.0
	
	
	
	IF #MessageNumber < 1 THEN //If message number 0 end function
	    RETURN;
	END_IF;
	
	
	
	IF  #MessageType= 'CNF' OR #MessageType = 'CNU' THEN
	    #MSG := #"_CNF_";
	ELSIF #MessageType = 'TRS' THEN
	    #MSG := #"_TRS_";
	ELSIF #MessageType = 'TRI' THEN
	    #MSG := #"_TRI_";
	ELSIF #MessageType = 'TRE' THEN
	    #MSG := #"_TRE_";
	ELSIF #MessageType = 'STA' THEN
	    #MSG := #"_STA_";
	ELSIF #MessageType = 'ANDON' THEN
	    #MSG := #"_ANDON_";
	ELSIF #MessageType = 'TRR' THEN
	    #MSG := #"_TRR_";
	ELSIF #MessageType = 'TRW' THEN
	    #MSG := #"_TRW_";
	ELSIF #MessageType = 'PFC' THEN
	    #MSG := #"_PFC_";
	ELSIF #MessageType = 'NFP' THEN
	    #MSG := #"_NFP_";
	ELSIF #MessageType = 'CMA' THEN
	    #MSG := #"_CMA_";
	ELSIF #MessageType = 'TMA' THEN
	    #MSG := #"_TMA_";
	ELSIF #MessageType = 'TRB' OR #MessageType = 'TRC' THEN
	    #MSG := #"_TRB_";
	    
	ELSE
	    RETURN;
	END_IF;
	
	IF NOT #SendMessage THEN // Error Reset
	    #State := 0;
	END_IF;
	
	#SEND_OFFSET.SW := (#MessageNumber * 2) + 2; //Calc message send sw offset
	#SEND_OFFSET.MSG := ((#MessageNumber - 1) * 80) + 604; // Calc send message offset
	#REC_OFFSET.SW := (#MessageNumber - 1) * 2; // Calc receive sw offset
	#REC_OFFSET.ANS := ((#MessageNumber - 1) * 32) + 600; // Calc receive answer offset
	#REC_OFFSET.MSG := ((#MessageNumber - 1) * 32) + 602; // Calc receive message offset
	
	
	CASE #State OF
	    0: // Initial State
	        #MessageDone := FALSE;
	        #Answer := 0;
	        #Fault := 0;
	        POKE(area := #DB, //Clear send flag
	             dbNumber := #DB_SEND,
	             byteOffset := #SEND_OFFSET.SW,
	             value := #MINUS1);
	        POKE(area := #DB, //Clear receive flag
	             dbNumber := #DB_REC,
	             byteOffset := #REC_OFFSET.SW,
	             value := #MINUS1);
	        #oNFP := #Blank;
	        #State := 10; ///Transition to state 10
	        
	    10: // Wait for start command
	        IF #SendMessage THEN //If start command active
	            //Clear NFP
	            #oNFP := #Blank;
	            
	            POKE(area := #DB, //Clear send flag
	                 dbNumber := #DB_SEND,
	                 byteOffset := #SEND_OFFSET.SW,
	                 value := #MINUS1);
	            POKE(area := #DB, //Clear receive flag
	                 dbNumber := #DB_REC,
	                 byteOffset := #REC_OFFSET.SW,
	                 value := #MINUS1);
	            POKE(area := #DB, // Clear answer 
	                 dbNumber := #DB_REC,
	                 byteOffset := #REC_OFFSET.ANS,
	                 value := #CLEAR);
	            
	            FOR #i := 0 TO 79 BY 1 DO //Clear all send array
	                POKE(area := #DB,
	                     dbNumber := #DB_SEND,
	                     byteOffset := (#SEND_OFFSET.MSG + #i),
	                     value := '$00');
	            END_FOR;
	            FOR #i := 0 TO 29 BY 1 DO //Clear all receive array
	                POKE(area := #DB,
	                     dbNumber := #DB_REC,
	                     byteOffset := (#REC_OFFSET.MSG + #i),
	                     value := '$00');
	            END_FOR;
	            #State := 20; //Transition to state 20
	        END_IF;
	        
	    20: // Create message to send
	        FOR #i := 0 TO 7 BY 1 DO //Copy NFP to DB to send
	            POKE(area := #DB,
	                 dbNumber := #DB_SEND,
	                 byteOffset := (#SEND_OFFSET.MSG + #i),
	                 value := #NFP[#i + 1]);
	        END_FOR;
	        CASE #MSG OF
	            #"_CNF_",#"_TRB_":
	                #CNT := (LEN(#Scan));
	                VAL_STRG(IN := #CNT,
	                         SIZE := 2,
	                         PREC := 0,
	                         FORMAT := W#16#0,
	                         P := 1,
	                         OUT => #CNT_STR);
	                IF #CNT < 10 THEN
	                    #CNT_STR := REPLACE(IN1 := #CNT_STR, IN2 := '0',
	                                        L := 1,
	                                        P := FIND(IN1 := #CNT_STR,
	                                                  IN2 := ' '));
	                END_IF;
	                POKE(area := #DB,
	                     dbNumber := #DB_SEND,
	                     byteOffset := (#SEND_OFFSET.MSG + 8),
	                     value := #CNT_STR[1]);
	                POKE(area := #DB,
	                     dbNumber := #DB_SEND,
	                     byteOffset := (#SEND_OFFSET.MSG + 9),
	                     value := #CNT_STR[2]);
	                FOR #i := 0 TO 70 BY 1 DO
	                    POKE(area := #DB,
	                         dbNumber := #DB_SEND,
	                         byteOffset := (#SEND_OFFSET.MSG + #i + 10),
	                         value := #Scan[#i + 1]);
	                END_FOR;
	                
	            #"_TRS_":
	                POKE(area := #DB,
	                     dbNumber := #DB_SEND,
	                     byteOffset := (#SEND_OFFSET.MSG + 8),
	                     value := USINT_TO_CHAR(#ProcessStatus + 48));
	                POKE(area := #DB,
	                     dbNumber := #DB_SEND,
	                     byteOffset := (#SEND_OFFSET.MSG + 9),
	                     value := INT_TO_CHAR(48));
	
	                //ANGLE
	                POKE(area := #DB,
	                     dbNumber := #DB_SEND,
	                     byteOffset := (#SEND_OFFSET.MSG + 10),
	                     value := #ScrewAngle);
	                //TORQUE BEFORE POINT
	                POKE(area := #DB,
	                     dbNumber := #DB_SEND,
	                     byteOffset := (#SEND_OFFSET.MSG + 12),
	                     value := #ScrewTorqueInt);
	                    
	                    //TORQUE AFTER POINT
	                    POKE(area := #DB,
	                         dbNumber := #DB_SEND,
	                         byteOffset := (#SEND_OFFSET.MSG + 14),
	                         value := #ScrewTorqueFloat);
	            
	            #"_TRI_":
	                POKE(area := #DB, //Set the process status of the message
	                     dbNumber := #DB_SEND,
	                     byteOffset := (#SEND_OFFSET.MSG + 8),
	                     value := USINT_TO_CHAR(#ProcessStatus + 48));
	                
	            #"_STA_":
	                FOR #i := 0 TO 7 BY 1 DO //Copy NFP to DB to send
	                    POKE(area := #DB,
	                         dbNumber := #DB_SEND,
	                         byteOffset := (#SEND_OFFSET.MSG + #i),
	                         value := #NFP[#i + 1]);
	                END_FOR;
	                    IF #MasterNFP THEN
	                        #oNFP := #NFP;
	                    END_IF;
	      
	                
	            #"_PFC_":
	                POKE(area := #DB,
	                     dbNumber := #DB_SEND,
	                     byteOffset := (#SEND_OFFSET.MSG + 8),
	                     value := '0');
	                POKE(area := #DB,
	                     dbNumber := #DB_SEND,
	                     byteOffset := (#SEND_OFFSET.MSG + 9),
	                     value := '8');
	                FOR #i := 0 TO 7 BY 1 DO
	                    POKE(area := #DB,
	                         dbNumber := #DB_SEND,
	                         byteOffset := (#SEND_OFFSET.MSG + #i + 10),
	                         value := #KANBAN[#i + 1]);
	                END_FOR;
	                
	                
	            #"_NFP_":
	                POKE(area := #DB,
	                     dbNumber := #DB_SEND,
	                     byteOffset := (#SEND_OFFSET.MSG),
	                     value := '0');
	                POKE(area := #DB,
	                     dbNumber := #DB_SEND,
	                     byteOffset := (#SEND_OFFSET.MSG + 1),
	                     value := '8');
	                FOR #i := 1 TO 8 BY 1 DO
	                    POKE(area := #DB,
	                         dbNumber := #DB_SEND,
	                         byteOffset := (#SEND_OFFSET.MSG + #i + 1),
	                         value := #KANBAN[#i]);
	                END_FOR;
	                
	            #"_CMA_",#"_TMA_":
	                FOR #i := 0 TO 7 BY 1 DO
	                    POKE(area := #DB,
	                         dbNumber := #DB_SEND,
	                         byteOffset := (#SEND_OFFSET.MSG + #i + 8),
	                         value := #Scan[#i + 1]);
	                END_FOR;
	        END_CASE;
	        #State := 30; // Transition to state 30
	        
	    30: //Set flag to "1" to inform that PLC is ready to send (DB5 Ó 1005)
	            POKE(area := #DB,//Set flag to "1" to inform that PLC is ready to send
	                 dbNumber := #DB_SEND,
	                 byteOffset := #SEND_OFFSET.SW,
	                 value := #PLUS1);
	           #State := 40; // Transition to state 40
	
	        
	    40: //Wait to IJCORE response with "-1"
	        IF (PEEK_WORD(area := #DB, dbNumber := #DB_SEND, byteOffset := #SEND_OFFSET.SW) = #MINUS1)
	        THEN
	            #State := 50; // Transition to state 50
	        END_IF;
	        
	    50: //Check if IJCORE have answer from DB Receive
	        IF (PEEK_WORD(area := #DB, dbNumber := #DB_REC, byteOffset := #REC_OFFSET.SW) = #PLUS1)
	        THEN
	            #Answer := PEEK_WORD(area := #DB, dbNumber := #DB_REC, byteOffset := #REC_OFFSET.ANS); //Copy answer from IJCORE
	            IF #Answer <> #PLUS1 THEN
	                #Fault := #Answer;
	            END_IF;
	            #State := 60; // Transition to state 100
	        END_IF;
	        
	    60: //Change Flag to "-1"
	        POKE(area := #DB, //Set "-1" to IJCORE
	                 dbNumber := #DB_REC,
	                 byteOffset := #REC_OFFSET.SW,
	                 value := #MINUS1);
	            #State := 100; // Transition to state 100
	       
	       
	        100: //Sequence done
	            CASE #TraceabilityMode OF
	                1:// Full traceability
	                    IF #Answer = 1 THEN
	                        #MessageDone := TRUE;
	                    ELSE
	                        #MessageDone := FALSE;
	                    END_IF;
	                2:// Traceability only
	                    #MessageDone := TRUE;
	            END_CASE;
	
	        IF NOT #SendMessage THEN
	            #State := 0; // Transition to state 0
	        END_IF;
	END_CASE;
	
	
	
	
	
	
	
END_FUNCTION_BLOCK

ORGANIZATION_BLOCK "stationOutputs"   // OB124, LAD, ProgramCycle
TITLE = "Main Program Sweep (Cycle)"
{ S7_Optimized_Access := 'TRUE' }
VERSION : 0.1
// stored: AutoNumber true, IsIECCheckEnabled false, SetENOAutomatically false
   VAR_INPUT
      Initial_Call : Bool;   // Initial call of this OB
      Remanence : Bool;   // =True, if remanent data are available
   END_VAR
   VAR_TEMP
      estopOK : Bool;
   END_VAR
BEGIN

REGION Network 1: PRESENT PARTS
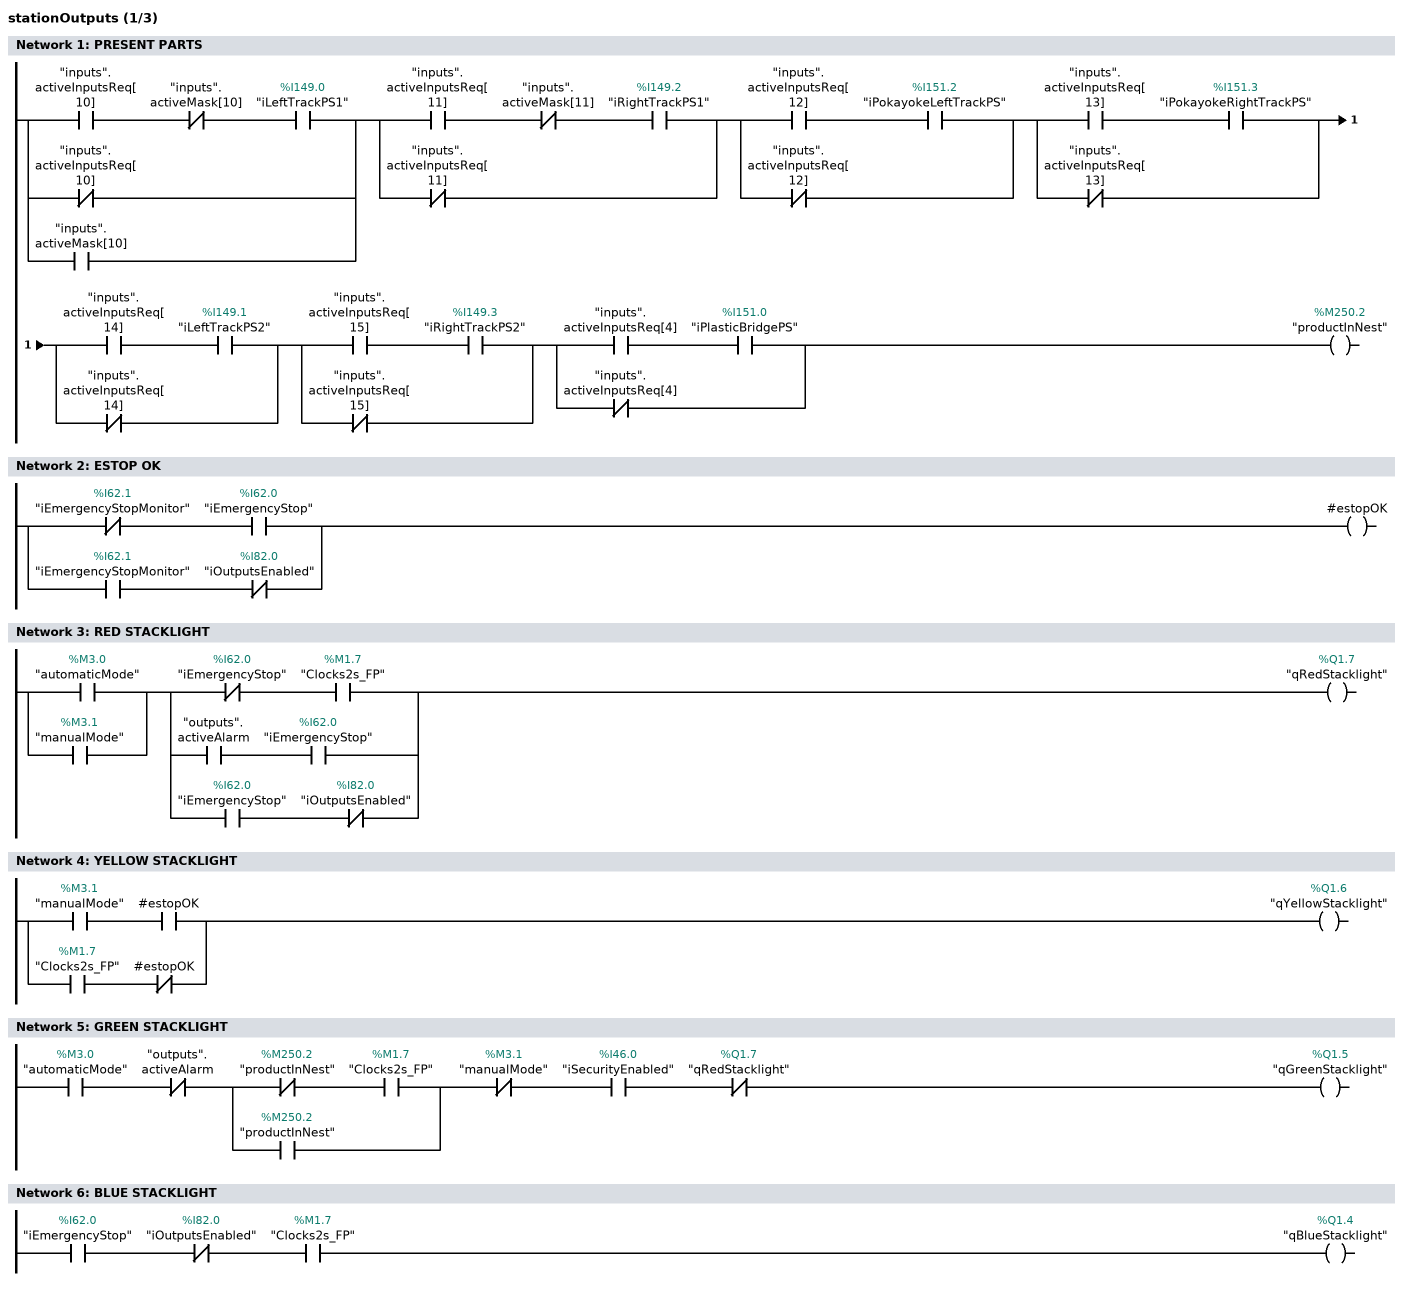
   RUNG wire#powerrail
      Contact( "inputs".activeInputsReq[10] )
      I_Contact( "inputs".activeMask[10] )
      Contact( "iLeftTrackPS1" )
      wire#w1
      Contact( "inputs".activeInputsReq[11] )
      I_Contact( "inputs".activeMask[11] )
      Contact( "iRightTrackPS1" )
      wire#w2
      Contact( "inputs".activeInputsReq[12] )
      Contact( "iPokayokeLeftTrackPS" )
      wire#w3
      Contact( "inputs".activeInputsReq[13] )
      Contact( "iPokayokeRightTrackPS" )
      wire#w4
      Contact( "inputs".activeInputsReq[14] )
      Contact( "iLeftTrackPS2" )
      wire#w5
      Contact( "inputs".activeInputsReq[15] )
      Contact( "iRightTrackPS2" )
      wire#w6
      Contact( "inputs".activeInputsReq[4] )
      Contact( "iPlasticBridgePS" )
      wire#w7
      Coil( "productInNest" )
   END_RUNG
   RUNG wire#powerrail
      I_Contact( "inputs".activeInputsReq[10] )
   END_RUNG wire#w1
   RUNG wire#powerrail
      Contact( "inputs".activeMask[10] )
   END_RUNG wire#w1
   RUNG wire#w1
      I_Contact( "inputs".activeInputsReq[11] )
   END_RUNG wire#w2
   RUNG wire#w2
      I_Contact( "inputs".activeInputsReq[12] )
   END_RUNG wire#w3
   RUNG wire#w3
      I_Contact( "inputs".activeInputsReq[13] )
   END_RUNG wire#w4
   RUNG wire#w4
      I_Contact( "inputs".activeInputsReq[14] )
   END_RUNG wire#w5
   RUNG wire#w5
      I_Contact( "inputs".activeInputsReq[15] )
   END_RUNG wire#w6
   RUNG wire#w6
      I_Contact( "inputs".activeInputsReq[4] )
   END_RUNG wire#w7
   // the same network as SCL:
   "productInNest" := (("inputs".activeInputsReq[10] AND NOT "inputs".activeMask[10] AND "iLeftTrackPS1") OR NOT "inputs".activeInputsReq[10] OR "inputs".activeMask[10]) AND (("inputs".activeInputsReq[11] AND NOT "inputs".activeMask[11] AND "iRightTrackPS1") OR NOT "inputs".activeInputsReq[11]) AND (("inputs".activeInputsReq[12] AND "iPokayokeLeftTrackPS") OR NOT "inputs".activeInputsReq[12]) AND (("inputs".activeInputsReq[13] AND "iPokayokeRightTrackPS") OR NOT "inputs".activeInputsReq[13]) AND (("inputs".activeInputsReq[14] AND "iLeftTrackPS2") OR NOT "inputs".activeInputsReq[14]) AND (("inputs".activeInputsReq[15] AND "iRightTrackPS2") OR NOT "inputs".activeInputsReq[15]) AND (("inputs".activeInputsReq[4] AND "iPlasticBridgePS") OR NOT "inputs".activeInputsReq[4]);
END_REGION

REGION Network 2: ESTOP OK
   RUNG wire#powerrail
      I_Contact( "iEmergencyStopMonitor" )
      Contact( "iEmergencyStop" )
      wire#w1
      Coil( #estopOK )
   END_RUNG
   RUNG wire#powerrail
      Contact( "iEmergencyStopMonitor" )
      I_Contact( "iOutputsEnabled" )
   END_RUNG wire#w1
   // the same network as SCL:
   #estopOK := (NOT "iEmergencyStopMonitor" AND "iEmergencyStop") OR ("iEmergencyStopMonitor" AND NOT "iOutputsEnabled");
END_REGION

REGION Network 3: RED STACKLIGHT
   RUNG wire#powerrail
      Contact( "automaticMode" )
      wire#w1
      I_Contact( "iEmergencyStop" )
      Contact( "Clocks2s_FP" )
      wire#w2
      Coil( "qRedStacklight" )
   END_RUNG
   RUNG wire#powerrail
      Contact( "manualMode" )
   END_RUNG wire#w1
   RUNG wire#w1
      Contact( "outputs".activeAlarm )
      Contact( "iEmergencyStop" )
   END_RUNG wire#w2
   RUNG wire#w1
      Contact( "iEmergencyStop" )
      I_Contact( "iOutputsEnabled" )
   END_RUNG wire#w2
   // the same network as SCL:
   "qRedStacklight" := ("automaticMode" OR "manualMode") AND ((NOT "iEmergencyStop" AND "Clocks2s_FP") OR ("outputs".activeAlarm AND "iEmergencyStop") OR ("iEmergencyStop" AND NOT "iOutputsEnabled"));
END_REGION

REGION Network 4: YELLOW STACKLIGHT
   RUNG wire#powerrail
      Contact( "manualMode" )
      Contact( #estopOK )
      wire#w1
      Coil( "qYellowStacklight" )
   END_RUNG
   RUNG wire#powerrail
      Contact( "Clocks2s_FP" )
      I_Contact( #estopOK )
   END_RUNG wire#w1
   // the same network as SCL:
   "qYellowStacklight" := ("manualMode" AND #estopOK) OR ("Clocks2s_FP" AND NOT #estopOK);
END_REGION

REGION Network 5: GREEN STACKLIGHT
   RUNG wire#powerrail
      Contact( "automaticMode" )
      I_Contact( "outputs".activeAlarm )
      wire#w1
      I_Contact( "productInNest" )
      Contact( "Clocks2s_FP" )
      wire#w2
      I_Contact( "manualMode" )
      Contact( "iSecurityEnabled" )
      I_Contact( "qRedStacklight" )
      Coil( "qGreenStacklight" )
   END_RUNG
   RUNG wire#w1
      Contact( "productInNest" )
   END_RUNG wire#w2
   // the same network as SCL:
   "qGreenStacklight" := "automaticMode" AND NOT "outputs".activeAlarm AND ((NOT "productInNest" AND "Clocks2s_FP") OR "productInNest") AND NOT "manualMode" AND "iSecurityEnabled" AND NOT "qRedStacklight";
END_REGION

REGION Network 6: BLUE STACKLIGHT
   RUNG wire#powerrail
      Contact( "iEmergencyStop" )
      I_Contact( "iOutputsEnabled" )
      Contact( "Clocks2s_FP" )
      Coil( "qBlueStacklight" )
   END_RUNG
   // the same network as SCL:
   "qBlueStacklight" := "iEmergencyStop" AND NOT "iOutputsEnabled" AND "Clocks2s_FP";
END_REGION

REGION Network 7: GREEN INDICATOR
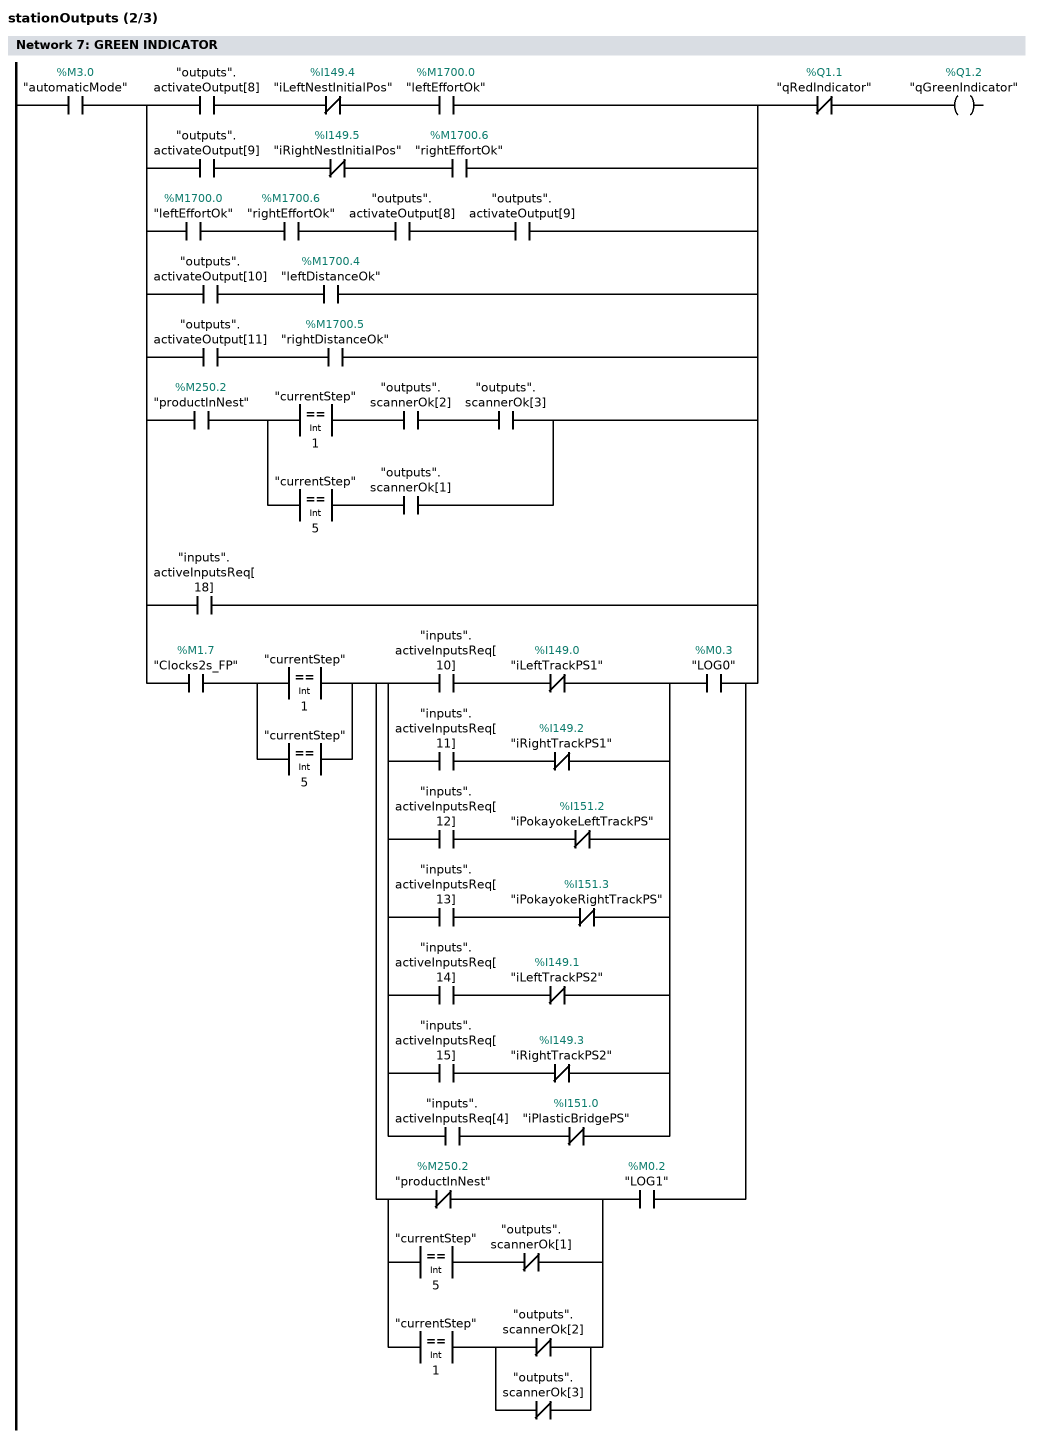
   RUNG wire#powerrail
      Contact( "automaticMode" )
      wire#w1
      Contact( "outputs".activateOutput[8] )
      I_Contact( "iLeftNestInitialPos" )
      Contact( "leftEffortOk" )
      wire#w2
      I_Contact( "qRedIndicator" )
      Coil( "qGreenIndicator" )
   END_RUNG
   RUNG wire#w1
      Contact( "outputs".activateOutput[9] )
      I_Contact( "iRightNestInitialPos" )
      Contact( "rightEffortOk" )
   END_RUNG wire#w2
   RUNG wire#w1
      Contact( "leftEffortOk" )
      Contact( "rightEffortOk" )
      Contact( "outputs".activateOutput[8] )
      Contact( "outputs".activateOutput[9] )
   END_RUNG wire#w2
   RUNG wire#w1
      Contact( "outputs".activateOutput[10] )
      Contact( "leftDistanceOk" )
   END_RUNG wire#w2
   RUNG wire#w1
      Contact( "outputs".activateOutput[11] )
      Contact( "rightDistanceOk" )
   END_RUNG wire#w2
   RUNG wire#w1
      Contact( "productInNest" )
      wire#w3
      { S7_Templates := "SrcType := Int" } EQ_Contact(in1 := "currentStep", in2 := 1)
      Contact( "outputs".scannerOk[2] )
      Contact( "outputs".scannerOk[3] )
   END_RUNG wire#w2
   RUNG wire#w3
      { S7_Templates := "SrcType := Int" } EQ_Contact(in1 := "currentStep", in2 := 5)
      Contact( "outputs".scannerOk[1] )
   END_RUNG wire#w2
   RUNG wire#w1
      Contact( "inputs".activeInputsReq[18] )
   END_RUNG wire#w2
   RUNG wire#w1
      Contact( "Clocks2s_FP" )
      wire#w4
      { S7_Templates := "SrcType := Int" } EQ_Contact(in1 := "currentStep", in2 := 1)
      wire#w5
      Contact( "inputs".activeInputsReq[10] )
      I_Contact( "iLeftTrackPS1" )
      wire#w6
      Contact( "LOG0" )
   END_RUNG wire#w2
   RUNG wire#w4
      { S7_Templates := "SrcType := Int" } EQ_Contact(in1 := "currentStep", in2 := 5)
   END_RUNG wire#w5
   RUNG wire#w5
      Contact( "inputs".activeInputsReq[11] )
      I_Contact( "iRightTrackPS1" )
   END_RUNG wire#w6
   RUNG wire#w5
      Contact( "inputs".activeInputsReq[12] )
      I_Contact( "iPokayokeLeftTrackPS" )
   END_RUNG wire#w6
   RUNG wire#w5
      Contact( "inputs".activeInputsReq[13] )
      I_Contact( "iPokayokeRightTrackPS" )
   END_RUNG wire#w6
   RUNG wire#w5
      Contact( "inputs".activeInputsReq[14] )
      I_Contact( "iLeftTrackPS2" )
   END_RUNG wire#w6
   RUNG wire#w5
      Contact( "inputs".activeInputsReq[15] )
      I_Contact( "iRightTrackPS2" )
   END_RUNG wire#w6
   RUNG wire#w5
      Contact( "inputs".activeInputsReq[4] )
      I_Contact( "iPlasticBridgePS" )
   END_RUNG wire#w6
   RUNG wire#w5
      I_Contact( "productInNest" )
      wire#w7
      Contact( "LOG1" )
   END_RUNG wire#w2
   RUNG wire#w5
      { S7_Templates := "SrcType := Int" } EQ_Contact(in1 := "currentStep", in2 := 5)
      I_Contact( "outputs".scannerOk[1] )
   END_RUNG wire#w7
   RUNG wire#w5
      { S7_Templates := "SrcType := Int" } EQ_Contact(in1 := "currentStep", in2 := 1)
      wire#w8
      I_Contact( "outputs".scannerOk[2] )
   END_RUNG wire#w7
   RUNG wire#w8
      I_Contact( "outputs".scannerOk[3] )
   END_RUNG wire#w7
   // the same network as SCL:
   "qGreenIndicator" := "automaticMode" AND (("outputs".activateOutput[8] AND NOT "iLeftNestInitialPos" AND "leftEffortOk") OR ("outputs".activateOutput[9] AND NOT "iRightNestInitialPos" AND "rightEffortOk") OR ("leftEffortOk" AND "rightEffortOk" AND "outputs".activateOutput[8] AND "outputs".activateOutput[9]) OR ("outputs".activateOutput[10] AND "leftDistanceOk") OR ("outputs".activateOutput[11] AND "rightDistanceOk") OR ("productInNest" AND ((("currentStep" = 1) AND "outputs".scannerOk[2] AND "outputs".scannerOk[3]) OR (("currentStep" = 5) AND "outputs".scannerOk[1]))) OR "inputs".activeInputsReq[18] OR ("Clocks2s_FP" AND (("currentStep" = 1) OR ("currentStep" = 5)) AND (((("inputs".activeInputsReq[10] AND NOT "iLeftTrackPS1") OR ("inputs".activeInputsReq[11] AND NOT "iRightTrackPS1") OR ("inputs".activeInputsReq[12] AND NOT "iPokayokeLeftTrackPS") OR ("inputs".activeInputsReq[13] AND NOT "iPokayokeRightTrackPS") OR ("inputs".activeInputsReq[14] AND NOT "iLeftTrackPS2") OR ("inputs".activeInputsReq[15] AND NOT "iRightTrackPS2") OR ("inputs".activeInputsReq[4] AND NOT "iPlasticBridgePS")) AND "LOG0") OR ((NOT "productInNest" OR (("currentStep" = 5) AND NOT "outputs".scannerOk[1]) OR (("currentStep" = 1) AND (NOT "outputs".scannerOk[2] OR NOT "outputs".scannerOk[3]))) AND "LOG1")))) AND NOT "qRedIndicator";
END_REGION

REGION Network 8: YELLOW INDICATOR
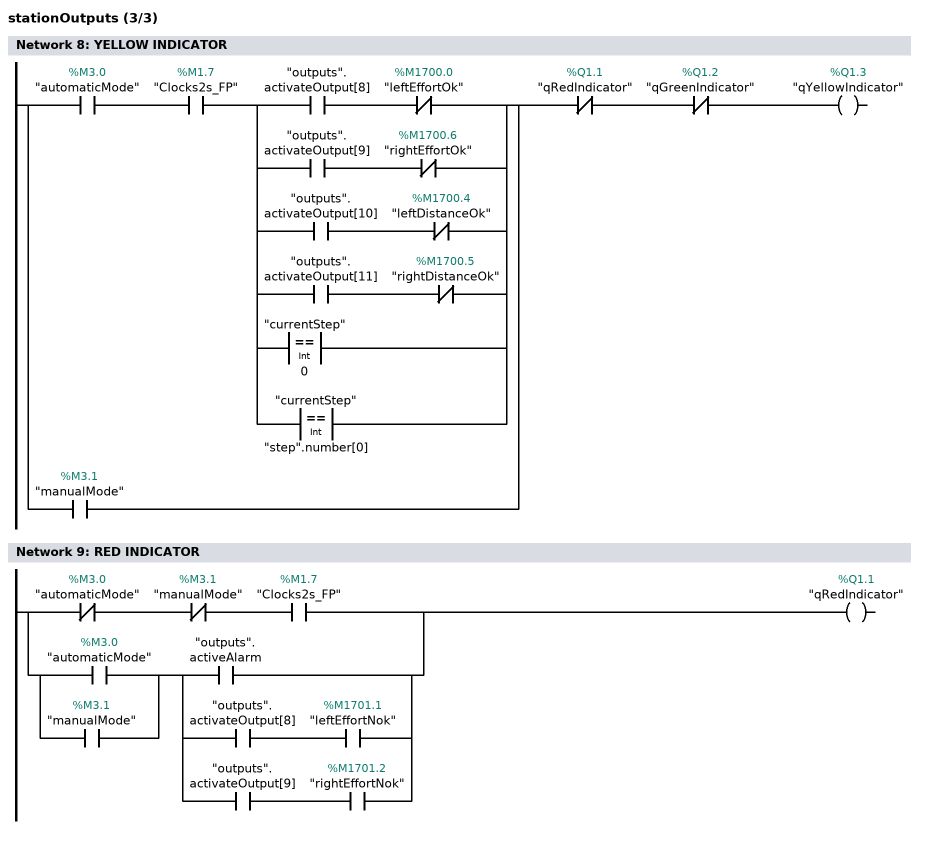
   RUNG wire#powerrail
      Contact( "automaticMode" )
      Contact( "Clocks2s_FP" )
      wire#w1
      Contact( "outputs".activateOutput[8] )
      I_Contact( "leftEffortOk" )
      wire#w2
      I_Contact( "qRedIndicator" )
      I_Contact( "qGreenIndicator" )
      Coil( "qYellowIndicator" )
   END_RUNG
   RUNG wire#w1
      Contact( "outputs".activateOutput[9] )
      I_Contact( "rightEffortOk" )
   END_RUNG wire#w2
   RUNG wire#w1
      Contact( "outputs".activateOutput[10] )
      I_Contact( "leftDistanceOk" )
   END_RUNG wire#w2
   RUNG wire#w1
      Contact( "outputs".activateOutput[11] )
      I_Contact( "rightDistanceOk" )
   END_RUNG wire#w2
   RUNG wire#w1
      { S7_Templates := "SrcType := Int" } EQ_Contact(in1 := "currentStep", in2 := 0)
   END_RUNG wire#w2
   RUNG wire#w1
      { S7_Templates := "SrcType := Int" } EQ_Contact(in1 := "currentStep", in2 := "step".number[0])
   END_RUNG wire#w2
   RUNG wire#powerrail
      Contact( "manualMode" )
   END_RUNG wire#w2
   // the same network as SCL:
   "qYellowIndicator" := (("automaticMode" AND "Clocks2s_FP" AND (("outputs".activateOutput[8] AND NOT "leftEffortOk") OR ("outputs".activateOutput[9] AND NOT "rightEffortOk") OR ("outputs".activateOutput[10] AND NOT "leftDistanceOk") OR ("outputs".activateOutput[11] AND NOT "rightDistanceOk") OR ("currentStep" = 0) OR ("currentStep" = "step".number[0]))) OR "manualMode") AND NOT "qRedIndicator" AND NOT "qGreenIndicator";
END_REGION

REGION Network 9: RED INDICATOR
   RUNG wire#powerrail
      I_Contact( "automaticMode" )
      I_Contact( "manualMode" )
      Contact( "Clocks2s_FP" )
      wire#w1
      Coil( "qRedIndicator" )
   END_RUNG
   RUNG wire#powerrail
      Contact( "automaticMode" )
      wire#w2
      Contact( "outputs".activeAlarm )
   END_RUNG wire#w1
   RUNG wire#powerrail
      Contact( "manualMode" )
   END_RUNG wire#w2
   RUNG wire#w2
      Contact( "outputs".activateOutput[8] )
      Contact( "leftEffortNok" )
   END_RUNG wire#w1
   RUNG wire#w2
      Contact( "outputs".activateOutput[9] )
      Contact( "rightEffortNok" )
   END_RUNG wire#w1
   // the same network as SCL:
   "qRedIndicator" := (NOT "automaticMode" AND NOT "manualMode" AND "Clocks2s_FP") OR (("automaticMode" OR "manualMode") AND ("outputs".activeAlarm OR ("outputs".activateOutput[8] AND "leftEffortNok") OR ("outputs".activateOutput[9] AND "rightEffortNok")));
END_REGION
END_ORGANIZATION_BLOCK

ORGANIZATION_BLOCK "sequence"
TITLE = "Main Program Sweep (Cycle)"
{ S7_Optimized_Access := 'TRUE' }
VERSION : 0.1
   VAR_TEMP 
      i : Int;
   END_VAR


BEGIN
	IF "automaticMode" = TRUE AND "currentModel" <> 0 AND "outputs".activeAlarm =  0 THEN
	    IF "currentStep" <= "step".number[0] THEN
	        
	        
	//***********************************************************************************************************************************************************************           
	//***********************************************************************************************************************************************************************                  
	                                               //****ENTRADAS****//
	                                            
	                                       
	        IF ("verificacion_estados_A" = 32) THEN
	                
	            "verificacion_estados_A" := 0;
	            "a_estados" := 0;
	            "a_correctas" := 0;
	                
	          END_IF;
	        
	        
	            IF "verificacion_estados_A" <= 31 THEN
	                
	// INICIO DE CONTEO DE LOS ESTADOS_A.
	                IF "inputs".inputActive["verificacion_estados_A"] = 1 AND "inputs".activeInputsReq["verificacion_estados_A"] = 0 AND "inputs".activeMask["verificacion_estados_A"] = 0 THEN
	                    "a_estados" := "a_estados" + 1;
	                END_IF;
	                
	                IF "inputs".activeInputsReq["verificacion_estados_A"] = 0 AND "inputs".activeMask["verificacion_estados_A"] = 1 THEN
	                    "a_estados" := "a_estados" + 1;
	                END_IF;
	                
	                IF "inputs".activeInputsReq["verificacion_estados_A"] = 1 AND "inputs".activeMask["verificacion_estados_A"] = 0 THEN
	                    "a_estados" := "a_estados" + 1;
	                END_IF;
	                
	                IF "inputs".activeInputsReq["verificacion_estados_A"] = 1 AND "inputs".activeMask["verificacion_estados_A"] = 1 THEN
	                    "a_estados" := "a_estados" + 1;
	                END_IF;
	// INICIO DE CONTEO DE TODOS LOS ESTADOS_A.
	                
	// INICIO DE CONTEO DE ESTADO DE ENTRADAS CORRECTAS.
	                IF "inputs".inputActive["verificacion_estados_A"] = 0 AND "inputs".activeInputsReq["verificacion_estados_A"] = 0 AND "inputs".activeMask["verificacion_estados_A"] = 1 THEN
	                    "a_correctas" := "a_correctas" + 1;
	                END_IF;
	                
	                IF "inputs".inputActive["verificacion_estados_A"] = 0 AND "inputs".activeInputsReq["verificacion_estados_A"] = 1 AND "inputs".activeMask["verificacion_estados_A"] = 1 THEN
	                    "a_correctas" := "a_correctas" + 1;
	                END_IF;
	                
	                IF "inputs".inputActive["verificacion_estados_A"] = 1 AND "inputs".activeInputsReq["verificacion_estados_A"] = 0 AND "inputs".activeMask["verificacion_estados_A"] = 1 THEN
	                    "a_correctas" := "a_correctas" + 1;
	                END_IF;
	                
	                IF "inputs".inputActive["verificacion_estados_A"] = 1 AND "inputs".activeInputsReq["verificacion_estados_A"] = 1 AND "inputs".activeMask["verificacion_estados_A"] = 0 THEN
	                    "a_correctas" := "a_correctas" + 1;
	                END_IF;
	                
	                IF "inputs".inputActive["verificacion_estados_A"] = 1 AND "inputs".activeInputsReq["verificacion_estados_A"] = 1 AND "inputs".activeMask["verificacion_estados_A"] = 1 THEN
	                    "a_correctas" := "a_correctas" + 1;
	                END_IF;
	// FIN DE CONTEO DE ESTADO DE ENTRADAS CORRECTAS.
	                
	                "verificacion_estados_A" := "verificacion_estados_A" + 1;
	            END_IF;
	            
	            
	//***********************************************************************************************************************************************************************           
	//***********************************************************************************************************************************************************************                  
	                                                        //****SALIDAS****//         
	                                                        
	            IF "verificacion_estados_B" = 32 THEN
	                
	                "verificacion_estados_B" := 0;
	                "b_estados" := 0;
	                "numberOfCorrectOutputStates" := 0;
	                
	            END_IF;
	            
	            IF "verificacion_estados_B" <= 31 THEN
	                
	// INICIO DE CONTEO DE LOS ESTADOS_B.
	                IF "outputs".outputsActive["verificacion_estados_B"] = 1 AND "outputs".activeOutputsReq["verificacion_estados_B"] = 0 AND "outputs".activeMask["verificacion_estados_B"] = 0 THEN
	                    "b_estados" := "b_estados" + 1;
	                END_IF;
	                
	                IF "outputs".activeOutputsReq["verificacion_estados_B"] = 0 AND "outputs".activeMask["verificacion_estados_B"] = 1 THEN
	                    "b_estados" := "b_estados" + 1;
	                END_IF;
	                
	                IF "outputs".activeOutputsReq["verificacion_estados_B"] = 1 AND "outputs".activeMask["verificacion_estados_B"] = 0 THEN
	                    "b_estados" := "b_estados" + 1;
	                END_IF;
	                
	                IF "outputs".activeOutputsReq["verificacion_estados_B"] = 1 AND "outputs".activeMask["verificacion_estados_B"] = 1 THEN
	                    "b_estados" := "b_estados" + 1;
	                END_IF;
	// FIN DE CONTEO DE TODOS LOS ESTADOS_B.
	                
	                
	// DESACTIVACIÓN DE SALIDA CUANDO NO ES REQUERIDA.
	                
	                IF "outputs".activeOutputsReq["verificacion_estados_B"] = 0 THEN
	                    "outputs".activateOutput["verificacion_estados_B"] := 0;
	                END_IF;
	                
	            
	// INICIO DE CONTEO DE ESTADO DE "SALIDAS" CORRECTAS.
	                IF "outputs".activeOutputsReq["verificacion_estados_B"] = 0 AND "outputs".activeMask["verificacion_estados_B"] = 1 THEN
	                    "numberOfCorrectOutputStates" := "numberOfCorrectOutputStates" + 1;
	                  
	                END_IF;
	                
	                IF "outputs".activeOutputsReq["verificacion_estados_B"] = 1 AND "outputs".activeMask["verificacion_estados_B"] = 1 THEN
	                    "outputs".activateOutput["verificacion_estados_B"] := 1;
	                    //IF "SALIDAS".TIMER ["verificacion_estados_B"].Q = 1 THEN
	                        "numberOfCorrectOutputStates" := "numberOfCorrectOutputStates" + 1;
	                    // END_IF;
	                END_IF;
	                
	                IF "outputs".activeOutputsReq["verificacion_estados_B"] = 1 AND "outputs".activeMask["verificacion_estados_B"] = 0 THEN
	                    "outputs".activateOutput["verificacion_estados_B"] := 1;
	                   // IF "SALIDAS".TIMER ["verificacion_estados_B"].Q = 1 THEN
	                        IF "outputs".outputsActive["verificacion_estados_B"] = 1 THEN
	                            "numberOfCorrectOutputStates" := "numberOfCorrectOutputStates" + 1;
	                        END_IF;
	                   //END_IF;
	                END_IF;
	                
	// FIN DE CONTEO DE ESTADO DE "SALIDAS" CORRECTAS.
	                
	                "verificacion_estados_B" := "verificacion_estados_B" + 1;
	            END_IF;
	            
	            
	                                                     
	//***********************************************************************************************************************************************************************           
	//***********************************************************************************************************************************************************************                  
	                                                     //****ENTRADAS****//
	                                                     
	            IF "outputs".showTextsOutputs = 0 THEN
	                
	                IF "aa" <= 31 THEN
	                    
	// INICIO DE COMPARACIONES DE DETECCIÓN DE SEÑALES DE ENTRADAS FALTANTES O SOBRANTES.  
	                    IF ("inputs".activeMask["aa"] = 1) OR (("inputs".activeInputsReq["aa"] = 1) AND ("inputs".inputActive["aa"] = 1)) OR (("inputs".activeInputsReq["aa"] = 0) AND ("inputs".inputActive["aa"] = 0)) THEN
	                        "aa" := "aa" + 1;
	                        IF "aa" = 32 THEN
	                            "aa" := 0;
	                            "outputs".showTextsOutputs := 1;
	                        END_IF;
	                    END_IF;
	                    
	                    IF ("inputs".activeMask["aa"] = 0) AND "inputs".activeInputsReq["aa"] = 1 AND "inputs".inputActive["aa"] = 0 THEN
	                        
	                        IF "allowedTextChange" = 0 THEN
	                            "hmi".operatorTextIndicator := CONCAT(IN1 := 'ESPERANDO POR ', IN2 := "inputs".inputText["aa"]);
	                            "aa" := "aa" + 1;
	                            IF "aa" = 32 THEN
	                                "aa" := 0;
	                                "outputs".showTextsOutputs := 1;
	                            END_IF;
	                        END_IF;
	                        
	                    END_IF;
	                    
	                    IF ("inputs".activeMask["aa"] = 0) AND "inputs".activeInputsReq["aa"] = 0 AND "inputs".inputActive["aa"] = 1 THEN
	                        
	                        IF "allowedTextChange" = 0 THEN
	                            "hmi".operatorTextIndicator := CONCAT(IN1 := 'ESPERANDO POR NO ', IN2 := "inputs".inputText["aa"]);
	                            "aa" := "aa" + 1;
	                            IF "aa" = 32 THEN
	                                "aa" := 0;
	                                "outputs".showTextsOutputs := 1;
	                            END_IF;
	                        END_IF;
	                        
	                    END_IF;
	//FIN DE COMPARACIONES DE DETECCIÓN DE SEÑALES DE ENTRADAS FALTANTES O SOBRANTES. 
	                    
	                    
	                END_IF;
	            END_IF;
	            
	        
	        
	//***********************************************************************************************************************************************************************           
	//***********************************************************************************************************************************************************************                  
	                                                    //****SALIDAS****//
	                                                   
	            IF "outputs".showTextsOutputs = 1 THEN
	                
	                IF "bb" <= 31 THEN
	                    
	// INICIO DE COMPARACIONES DE DETECCIÓN DE SEÑALES DE SALIDAS FALTANTES O SOBRANTES.  
	                    IF ("outputs".activeMask["bb"] = 1) OR (("outputs".activeOutputsReq["bb"] = 1) AND ("outputs".outputsActive["bb"] = 1)) OR (("outputs".activeOutputsReq["bb"] = 0) AND ("outputs".outputsActive["bb"] = 0)) THEN
	                        "bb" := "bb" + 1;
	                        IF "bb" = 32 THEN
	                           "bb" := 0;
	                           "outputs".showTextsOutputs := 0;
	                        END_IF;
	                    END_IF;
	                    
	                    IF ("outputs".activeMask["bb"] = 0) AND "outputs".activeOutputsReq["bb"] = 1 AND "outputs".outputsActive["bb"] = 0 THEN
	                        
	                        IF "allowedTextChange" = 0 THEN
	                            "hmi".operatorTextIndicator := CONCAT(IN1 := 'ESPERANDO POR ', IN2 := "outputs".text["bb"]);
	                            "bb" := "bb" + 1;
	                            IF "bb" = 32 THEN
	                                "bb" := 0;
	                                "outputs".showTextsOutputs := 0;
	                            END_IF;
	                        END_IF;
	                        
	                    END_IF;
	                    
	                    IF ("outputs".activeMask["bb"] = 0) AND "outputs".activeOutputsReq["bb"] = 0 AND "outputs".outputsActive["bb"] = 1 THEN
	                        
	                        IF "allowedTextChange" = 0 THEN
	                            "hmi".operatorTextIndicator := CONCAT(IN1 := 'ESPERANDO POR NO ', IN2 := "outputs".text["bb"]);
	                            "bb" := "bb" + 1;
	                            IF "bb" = 32 THEN
	                                "bb" := 0;
	                                "outputs".showTextsOutputs := 0;
	                            END_IF;
	                        END_IF;
	                        
	                    END_IF;
	// FIN DE COMPARACIONES DE DETECCIÓN DE SEÑALES DE SALIDAS FALTANTES O SOBRANTES. 
	
	                END_IF;
	            END_IF;
	                                                    
	                                                    
	                                                    
	//***********************************************************************************************************************************************************************           
	//***********************************************************************************************************************************************************************                  
	                                                    //****CAMBIO DE PASO****//
	                                                    
	                                                    
	               
	            IF (("a_correctas" = "a_estados") AND ("a_correctas" <> 0) AND ("a_estados" <> 0) AND ("numberOfCorrectOutputStates" = "b_estados") AND ("numberOfCorrectOutputStates" <> 0) AND ("b_estados" <> 0) AND ("verificacion_estados_B" = 32) AND ("verificacion_estados_A" = 32)) OR (("inputs".inputSequence[0, "currentStep"] = 0) AND ("inputs".maskSequence[0, "currentStep"] = 0) AND ("inputs".activeInputsReqDInt = 0) AND ("verificacion_estados_A" = 32)) OR (("a_correctas" = "a_estados") AND ("a_correctas" <> 0) AND ("a_estados" <> 0) AND ("verificacion_estados_A" = 32) AND ("outputs".outputSequence[0, "currentStep"] = 0) AND ("outputs".maskSequence[0, "currentStep"] = 0) AND ("outputs".active = 0)) THEN
	                
	                "hmi".operatorTextIndicator := ' ';
	                
	                "step".stepChangeTimerStart := 1;
	                
	                IF "step".counterDone = 1 THEN
	                    "step".stepChangeTimerStart := 0;
	                END_IF;
	                
	                IF ("step".counterDone = 1 OR "step".stepChangeTimer = 0) THEN
	                    
	                    IF "currentStep" = "step".number[0] THEN
	                        IF "currentStep" <> 0 AND "step".number[0] <> 0 THEN
	                            "hmi".cicles := "hmi".cicles + 1;
	                            
	                            IF "shift1" THEN
	                                "hmi".production1 := "hmi".production1 + 1;
	                            END_IF;
	                            
	                            IF "shift2" THEN
	                                "hmi".production2 := "hmi".production2 + 1;
	                            END_IF;
	                            
	                            IF "shift3" THEN
	                                "hmi".production3 := "hmi".production3 + 1;
	                            END_IF;
	                            
	                            
	                        END_IF;
	                        "currentStep" := 0;
	                        RETURN;
	                    END_IF;
	                    
	                    "currentStep" := "currentStep" + 1;
	                   
	                END_IF;
	                
	                
	            END_IF;
	            
	            
	            
	        END_IF;
	      END_IF;
	      
	      
END_ORGANIZATION_BLOCK

DATA_BLOCK "FC_IJCORE_MAIN_DB"   // DB1000
VERSION : 0.1
// stored: AutoNumber false, DBAccessibleFromOPCUA true, DBAccessibleFromWebserver true, InstanceOfName FC_IJCORE_MAIN, InstanceOfType FB
"FC_IJCORE_MAIN"
BEGIN
   NFP[1..5] := '';
   AWK.ack_error := TRUE;
   AWK.State_com := 1;
   AWK.T1PresetValue := T#1S;
   AWK.T2PresetValue := T#1M;
   AWK.AwSignalTimeOutFault := FALSE;
   AWK.Reset_Counters := FALSE;
   AWK.Restart_Counter_bit_of_life := 4;
   AWK.NB_Bit_of_Life := FALSE;
   AWK.number_restart := 21346;
   AWK.check_restart := TRUE;
   AWK."Timer"[1].PT := T#1S;
   AWK."Timer"[2].PT := T#2S;
   AWK."Timer"[3].PT := T#200MS;
   AWK."Timer"[4].PT := T#1M;
   AWK."Timer"[5].PT := T#0MS;
   AWK."Timer"[1..3].IN := FALSE;
   AWK."Timer"[4].IN := TRUE;
   AWK."Timer"[5].IN := FALSE;
   MSG[1].MessageType := 'NFP';
   MSG[2..4].MessageType := 'TRC';
   MSG[5].MessageType := 'TRI';
   MSG[6..8].MessageType := 'CNF';
   MSG[9..20].MessageType := '';
   MSG[1].MessageNumber := 1;
   MSG[2].MessageNumber := 2;
   MSG[3].MessageNumber := 3;
   MSG[4].MessageNumber := 4;
   MSG[5].MessageNumber := 5;
   MSG[6].MessageNumber := 6;
   MSG[7].MessageNumber := 7;
   MSG[8].MessageNumber := 8;
   MSG[9..20].MessageNumber := 0;
   MSG[1..8].TraceabilityMode := 1;
   MSG[9..20].TraceabilityMode := 0;
   MSG[1..20].SendMessage := FALSE;
   MSG[1].MasterNFP := FALSE;
   MSG[2].MasterNFP := TRUE;
   MSG[3..20].MasterNFP := FALSE;
   MSG[1..20].NFP := '';
   MSG[1..20].Scan := '';
   MSG[1..20].KANBAN := '';
   MSG[1..20].ScrewTorqueInt := 16#0000;
   MSG[1..20].ScrewTorqueFloat := 16#0000;
   MSG[1..20].ScrewAngle := 16#0000;
   MSG[1..20].ProcessStatus := 0;
   MSG[1..8].ErrReset := TRUE;
   MSG[9..20].ErrReset := FALSE;
   MSG[1..20].oNFP := '';
   MSG[1..20].MessageDone := FALSE;
   MSG[1..20].Answer := 0;
   MSG[1..20].Fault := 0;
   MSG[1..8].State := 10;
   MSG[9..20].State := 0;
   MSG[1].SEND_OFFSET.SW := 4;
   MSG[2].SEND_OFFSET.SW := 6;
   MSG[3].SEND_OFFSET.SW := 8;
   MSG[4].SEND_OFFSET.SW := 10;
   MSG[5].SEND_OFFSET.SW := 12;
   MSG[6].SEND_OFFSET.SW := 14;
   MSG[7].SEND_OFFSET.SW := 16;
   MSG[8].SEND_OFFSET.SW := 18;
   MSG[9..20].SEND_OFFSET.SW := 0;
   MSG[1].SEND_OFFSET.MSG := 604;
   MSG[2].SEND_OFFSET.MSG := 684;
   MSG[3].SEND_OFFSET.MSG := 764;
   MSG[4].SEND_OFFSET.MSG := 844;
   MSG[5].SEND_OFFSET.MSG := 924;
   MSG[6].SEND_OFFSET.MSG := 1004;
   MSG[7].SEND_OFFSET.MSG := 1084;
   MSG[8].SEND_OFFSET.MSG := 1164;
   MSG[9..20].SEND_OFFSET.MSG := 0;
   MSG[1].REC_OFFSET.SW := 0;
   MSG[2].REC_OFFSET.SW := 2;
   MSG[3].REC_OFFSET.SW := 4;
   MSG[4].REC_OFFSET.SW := 6;
   MSG[5].REC_OFFSET.SW := 8;
   MSG[6].REC_OFFSET.SW := 10;
   MSG[7].REC_OFFSET.SW := 12;
   MSG[8].REC_OFFSET.SW := 14;
   MSG[9..20].REC_OFFSET.SW := 0;
   MSG[1].REC_OFFSET.MSG := 602;
   MSG[2].REC_OFFSET.MSG := 634;
   MSG[3].REC_OFFSET.MSG := 666;
   MSG[4].REC_OFFSET.MSG := 698;
   MSG[5].REC_OFFSET.MSG := 730;
   MSG[6].REC_OFFSET.MSG := 762;
   MSG[7].REC_OFFSET.MSG := 794;
   MSG[8].REC_OFFSET.MSG := 826;
   MSG[9..20].REC_OFFSET.MSG := 0;
   MSG[1].REC_OFFSET.ANS := 600;
   MSG[2].REC_OFFSET.ANS := 632;
   MSG[3].REC_OFFSET.ANS := 664;
   MSG[4].REC_OFFSET.ANS := 696;
   MSG[5].REC_OFFSET.ANS := 728;
   MSG[6].REC_OFFSET.ANS := 760;
   MSG[7].REC_OFFSET.ANS := 792;
   MSG[8].REC_OFFSET.ANS := 824;
   MSG[9..20].REC_OFFSET.ANS := 0;
   MSG[1].ONS[1..8] := FALSE;
   MSG[2].ONS[1..8] := FALSE;
   MSG[3].ONS[1..8] := FALSE;
   MSG[4].ONS[1..8] := FALSE;
   MSG[5].ONS[1..8] := FALSE;
   MSG[6].ONS[1..8] := FALSE;
   MSG[7].ONS[1..8] := FALSE;
   MSG[8].ONS[1..8] := FALSE;
   MSG[9].ONS[1..8] := FALSE;
   MSG[10].ONS[1..8] := FALSE;
   MSG[11].ONS[1..8] := FALSE;
   MSG[12].ONS[1..8] := FALSE;
   MSG[13].ONS[1..8] := FALSE;
   MSG[14].ONS[1..8] := FALSE;
   MSG[15].ONS[1..8] := FALSE;
   MSG[16].ONS[1..8] := FALSE;
   MSG[17].ONS[1..8] := FALSE;
   MSG[18].ONS[1..8] := FALSE;
   MSG[19].ONS[1..8] := FALSE;
   MSG[20].ONS[1..8] := FALSE;
   Faults[0..1] := 16#0000;
END_DATA_BLOCK

DATA_BLOCK "timeSystemDB"   // DB32
VERSION : 0.1
// stored: AutoNumber true, DBAccessibleFromOPCUA true, DBAccessibleFromWebserver true, InstanceOfName timeSystem, InstanceOfType FB
"timeSystem"
BEGIN
   nCycleTimeArray[0..5] := 0.0;
   tCycleTime.PT := T#0MS;
   tCycleTime.IN := FALSE;
   timesCounter.CU := FALSE;
   timesCounter.CD := FALSE;
   timesCounter.R := FALSE;
   timesCounter.LD := FALSE;
   timesCounter.QU := FALSE;
   timesCounter.QD := FALSE;
   timesCounter.PV := 5;
   timesCounter.CV := 0;
END_DATA_BLOCK

DATA_BLOCK "BUTTON SHUTOFF TIME"   // DB8
{ S7_Optimized_Access := 'TRUE' }
// stored: AutoNumber true, DBAccessibleFromOPCUA true, DBAccessibleFromWebserver true, InstanceOfName IEC_TIMER, OfSystemLibElement IEC_TIMER, OfSystemLibVersion 1.0
"IEC_TIMER"
   // VAR
   //    PT : Time := T#0MS;
   //    ET { ExternalWritable := 'False'} : Time;
   //    IN : Bool := FALSE;
   //    Q { ExternalWritable := 'False'} : Bool;
   // END_VAR
BEGIN
END_DATA_BLOCK

DATA_BLOCK "CYL 10 DIR A TON"   // DB50
{ S7_Optimized_Access := 'TRUE' }
// stored: AutoNumber true, DBAccessibleFromOPCUA true, DBAccessibleFromWebserver true, InstanceOfName IEC_TIMER, OfSystemLibElement IEC_TIMER, OfSystemLibVersion 1.0
"IEC_TIMER"
   // VAR
   //    PT : Time := T#0MS;
   //    ET { ExternalWritable := 'False'} : Time;
   //    IN : Bool := FALSE;
   //    Q { ExternalWritable := 'False'} : Bool;
   // END_VAR
BEGIN
END_DATA_BLOCK

DATA_BLOCK "CYL 10 DIR B TON"   // DB52
{ S7_Optimized_Access := 'TRUE' }
// stored: AutoNumber true, DBAccessibleFromOPCUA true, DBAccessibleFromWebserver true, InstanceOfName IEC_TIMER, OfSystemLibElement IEC_TIMER, OfSystemLibVersion 1.0
"IEC_TIMER"
   // VAR
   //    PT : Time := T#0MS;
   //    ET { ExternalWritable := 'False'} : Time;
   //    IN : Bool := FALSE;
   //    Q { ExternalWritable := 'False'} : Bool;
   // END_VAR
BEGIN
END_DATA_BLOCK

DATA_BLOCK "DIRECTION PULSE CTU"   // DB23
{ S7_Optimized_Access := 'TRUE' }
// stored: AutoNumber true, DBAccessibleFromOPCUA true, DBAccessibleFromWebserver true, InstanceOfName IEC_COUNTER, OfSystemLibElement IEC_COUNTER, OfSystemLibVersion 1.0
"IEC_COUNTER"
   // VAR RETAIN
   //    CU : Bool := FALSE;
   //    CD : Bool := FALSE;
   //    R : Bool := FALSE;
   //    LD : Bool := FALSE;
   //    QU : Bool := FALSE;
   //    QD : Bool := FALSE;
   //    PV : Int := 10;
   //    CV : Int := 2;
   // END_VAR
BEGIN
END_DATA_BLOCK

DATA_BLOCK "FC_EKS_R_TRIG_0"   // DB8200
// stored: AutoNumber true, DBAccessibleFromOPCUA true, DBAccessibleFromWebserver true, InstanceOfName R_TRIG, OfSystemLibElement R_TRIG, OfSystemLibVersion 1.0
"R_TRIG"
   // VAR_INPUT
   //    CLK : Bool := FALSE;
   // END_VAR
   // VAR_OUTPUT
   //    Q : Bool := FALSE;
   // END_VAR
   // VAR
   //    Stat_Bit : Bool := FALSE;
   // END_VAR
BEGIN
END_DATA_BLOCK

DATA_BLOCK "IEC_Timer_0_DB"   // DB13
{ S7_Optimized_Access := 'TRUE' }
// stored: AutoNumber true, DBAccessibleFromOPCUA true, DBAccessibleFromWebserver true, InstanceOfName IEC_TIMER, OfSystemLibElement IEC_TIMER, OfSystemLibVersion 1.0
"IEC_TIMER"
   // VAR
   //    PT : Time := T#2S;
   //    ET { ExternalWritable := 'False'} : Time;
   //    IN : Bool := FALSE;
   //    Q { ExternalWritable := 'False'} : Bool;
   // END_VAR
BEGIN
END_DATA_BLOCK

DATA_BLOCK "IEC_Timer_0_DB_1"   // DB64
{ S7_Optimized_Access := 'TRUE' }
// stored: AutoNumber true, DBAccessibleFromOPCUA true, DBAccessibleFromWebserver true, InstanceOfName IEC_TIMER, OfSystemLibElement IEC_TIMER, OfSystemLibVersion 1.0
"IEC_TIMER"
   // VAR
   //    PT : Time := T#1M_40S;
   //    ET { ExternalWritable := 'False'} : Time;
   //    IN : Bool := FALSE;
   //    Q { ExternalWritable := 'False'} : Bool;
   // END_VAR
BEGIN
END_DATA_BLOCK

DATA_BLOCK "IEC_Timer_0_DB_3"   // DB14
{ S7_Optimized_Access := 'TRUE' }
// stored: AutoNumber true, DBAccessibleFromOPCUA true, DBAccessibleFromWebserver true, InstanceOfName IEC_TIMER, OfSystemLibElement IEC_TIMER, OfSystemLibVersion 1.0
"IEC_TIMER"
   // VAR
   //    PT : Time := T#2S;
   //    ET { ExternalWritable := 'False'} : Time;
   //    IN : Bool := FALSE;
   //    Q { ExternalWritable := 'False'} : Bool;
   // END_VAR
BEGIN
END_DATA_BLOCK

DATA_BLOCK "IEC_Timer_0_DB_4"   // DB20
{ S7_Optimized_Access := 'TRUE' }
// stored: AutoNumber true, DBAccessibleFromOPCUA true, DBAccessibleFromWebserver true, InstanceOfName IEC_TIMER, OfSystemLibElement IEC_TIMER, OfSystemLibVersion 1.0
"IEC_TIMER"
   // VAR
   //    PT : Time := T#2S;
   //    ET { ExternalWritable := 'False'} : Time;
   //    IN : Bool := FALSE;
   //    Q { ExternalWritable := 'False'} : Bool;
   // END_VAR
BEGIN
END_DATA_BLOCK

DATA_BLOCK "IEC_Timer_0_DB_5"   // DB21
{ S7_Optimized_Access := 'TRUE' }
// stored: AutoNumber true, DBAccessibleFromOPCUA true, DBAccessibleFromWebserver true, InstanceOfName IEC_TIMER, OfSystemLibElement IEC_TIMER, OfSystemLibVersion 1.0
"IEC_TIMER"
   // VAR
   //    PT : Time := T#2S;
   //    ET { ExternalWritable := 'False'} : Time;
   //    IN : Bool := FALSE;
   //    Q { ExternalWritable := 'False'} : Bool;
   // END_VAR
BEGIN
END_DATA_BLOCK

DATA_BLOCK "IEC_Timer_0_DB_6"   // DB24
{ S7_Optimized_Access := 'TRUE' }
// stored: AutoNumber true, DBAccessibleFromOPCUA true, DBAccessibleFromWebserver true, InstanceOfName IEC_TIMER, OfSystemLibElement IEC_TIMER, OfSystemLibVersion 1.0
"IEC_TIMER"
   // VAR
   //    PT : Time := T#2S;
   //    ET { ExternalWritable := 'False'} : Time;
   //    IN : Bool := FALSE;
   //    Q { ExternalWritable := 'False'} : Bool;
   // END_VAR
BEGIN
END_DATA_BLOCK

DATA_BLOCK "IEC_Timer_0_DB_7"   // DB25
{ S7_Optimized_Access := 'TRUE' }
// stored: AutoNumber true, DBAccessibleFromOPCUA true, DBAccessibleFromWebserver true, InstanceOfName IEC_TIMER, OfSystemLibElement IEC_TIMER, OfSystemLibVersion 1.0
"IEC_TIMER"
   // VAR
   //    PT : Time := T#2S;
   //    ET { ExternalWritable := 'False'} : Time;
   //    IN : Bool := FALSE;
   //    Q { ExternalWritable := 'False'} : Bool;
   // END_VAR
BEGIN
END_DATA_BLOCK

DATA_BLOCK "IEC_Timer_0_DB_8"   // DB26
{ S7_Optimized_Access := 'TRUE' }
// stored: AutoNumber true, DBAccessibleFromOPCUA true, DBAccessibleFromWebserver true, InstanceOfName IEC_TIMER, OfSystemLibElement IEC_TIMER, OfSystemLibVersion 1.0
"IEC_TIMER"
   // VAR
   //    PT : Time := T#2S;
   //    ET { ExternalWritable := 'False'} : Time;
   //    IN : Bool := FALSE;
   //    Q { ExternalWritable := 'False'} : Bool;
   // END_VAR
BEGIN
END_DATA_BLOCK

DATA_BLOCK "IEC_Timer_0_DB_9"   // DB27
{ S7_Optimized_Access := 'TRUE' }
// stored: AutoNumber true, DBAccessibleFromOPCUA true, DBAccessibleFromWebserver true, InstanceOfName IEC_TIMER, OfSystemLibElement IEC_TIMER, OfSystemLibVersion 1.0
"IEC_TIMER"
   // VAR
   //    PT : Time := T#2S;
   //    ET { ExternalWritable := 'False'} : Time;
   //    IN : Bool := FALSE;
   //    Q { ExternalWritable := 'False'} : Bool;
   // END_VAR
BEGIN
END_DATA_BLOCK

DATA_BLOCK "OPERATOR TEXT INDICATOR TIMER"   // DB9
{ S7_Optimized_Access := 'TRUE' }
// stored: AutoNumber true, DBAccessibleFromOPCUA true, DBAccessibleFromWebserver true, InstanceOfName IEC_TIMER, OfSystemLibElement IEC_TIMER, OfSystemLibVersion 1.0
"IEC_TIMER"
   // VAR
   //    PT : Time := T#800MS;
   //    ET { ExternalWritable := 'False'} : Time;
   //    IN : Bool := FALSE;
   //    Q { ExternalWritable := 'False'} : Bool;
   // END_VAR
BEGIN
END_DATA_BLOCK

DATA_BLOCK "PERIODO_TON"   // DB18
{ S7_Optimized_Access := 'TRUE' }
// stored: AutoNumber true, DBAccessibleFromOPCUA true, DBAccessibleFromWebserver true, InstanceOfName IEC_TIMER, OfSystemLibElement IEC_TIMER, OfSystemLibVersion 1.0
"IEC_TIMER"
   // VAR
   //    PT : Time := T#200MS;
   //    ET { ExternalWritable := 'False'} : Time;
   //    IN : Bool := FALSE;
   //    Q { ExternalWritable := 'False'} : Bool;
   // END_VAR
BEGIN
END_DATA_BLOCK

DATA_BLOCK "PREASSURE_SENSOR_TIMER"   // DB16
{ S7_Optimized_Access := 'TRUE' }
// stored: AutoNumber true, DBAccessibleFromOPCUA true, DBAccessibleFromWebserver true, InstanceOfName IEC_TIMER, OfSystemLibElement IEC_TIMER, OfSystemLibVersion 1.0
"IEC_TIMER"
   // VAR
   //    PT : Time := T#3S;
   //    ET { ExternalWritable := 'False'} : Time;
   //    IN : Bool := FALSE;
   //    Q { ExternalWritable := 'False'} : Bool;
   // END_VAR
BEGIN
END_DATA_BLOCK

DATA_BLOCK "PULSE CTU"   // DB22
{ S7_Optimized_Access := 'TRUE' }
// stored: AutoNumber true, DBAccessibleFromOPCUA true, DBAccessibleFromWebserver true, InstanceOfName IEC_COUNTER, OfSystemLibElement IEC_COUNTER, OfSystemLibVersion 1.0
"IEC_COUNTER"
   // VAR RETAIN
   //    CU : Bool := FALSE;
   //    CD : Bool := FALSE;
   //    R : Bool := FALSE;
   //    LD : Bool := FALSE;
   //    QU : Bool := FALSE;
   //    QD : Bool := FALSE;
   //    PV : Int := 5;
   //    CV : Int := 2;
   // END_VAR
BEGIN
END_DATA_BLOCK

DATA_BLOCK "PULSO ALTO"   // DB15
{ S7_Optimized_Access := 'TRUE' }
// stored: AutoNumber true, DBAccessibleFromOPCUA true, DBAccessibleFromWebserver true, InstanceOfName IEC_TIMER, OfSystemLibElement IEC_TIMER, OfSystemLibVersion 1.0
"IEC_TIMER"
   // VAR
   //    PT : Time := T#10MS;
   //    ET { ExternalWritable := 'False'} : Time;
   //    IN : Bool := FALSE;
   //    Q { ExternalWritable := 'False'} : Bool;
   // END_VAR
BEGIN
END_DATA_BLOCK

DATA_BLOCK "Port_Config_DB2"   // DB38
// stored: AutoNumber true, DBAccessibleFromOPCUA true, DBAccessibleFromWebserver true, InstanceOfName Port_Config, OfSystemLibElement Port_Config, OfSystemLibVersion 1.2
"Port_Config"
   // VAR_INPUT
   //    REQ : Bool := TRUE;
   //    PORT : PORT := 284;
   //    PROTOCOL : UInt := 0;
   //    BAUD : UInt := 6;
   //    PARITY : UInt := 1;
   //    DATABITS : UInt := 1;
   //    STOPBITS : UInt := 1;
   //    FLOWCTRL : UInt := 2;
   //    XONCHAR : Char := '$0B';
   //    XOFFCHAR : Char := '$R';
   //    WAITTIME : UInt := 2000;
   //    MODE : USInt := 0;
   //    LINE_PRE : USInt := 0;
   //    BRK_DET : USInt := 0;
   // END_VAR
   // VAR_OUTPUT
   //    DONE : Bool := FALSE;
   //    ERROR : Bool := FALSE;
   //    STATUS : Word := 16#7000;
   // END_VAR
   // VAR
   //    b_e_REQ : Bool := TRUE;
   //    y_state : SInt := 0;
   //    WRREC { S7_SetPoint := 'True'} : WRREC;
   //    RDREC { S7_SetPoint := 'True'} : RDREC;
   //    w_record { S7_SetPoint := 'True'} : P2P_PortData;
   //    r_record { S7_SetPoint := 'True'} : P2P_RdEstat;
   // END_VAR
BEGIN
   WRREC.REQ := FALSE;
   WRREC.ID := 284;
   WRREC.INDEX := 57;
   WRREC.LEN := 28;
   WRREC.DONE := TRUE;
   WRREC.BUSY := FALSE;
   WRREC.ERROR := FALSE;
   WRREC.STATUS := 16#0000_0000;
   RDREC.REQ := FALSE;
   RDREC.ID := 0;
   RDREC.INDEX := 0;
   RDREC.MLEN := 0;
   RDREC.VALID := FALSE;
   RDREC.BUSY := FALSE;
   RDREC.ERROR := FALSE;
   RDREC.STATUS := 16#0000_0000;
   RDREC.LEN := 0;
   w_record.header.block_type := 16#0039;
   w_record.header.block_len := 16#0018;
   w_record.header.block_ver := 16#0100;
   w_record.header.res := 16#0000;
   w_record.PROTOCOL := 0;
   w_record.BAUD := 6;
   w_record.PARITY := 1;
   w_record.DATABITS := 1;
   w_record.STOPBITS := 1;
   w_record.FLOWCTRL := 2;
   w_record.XONCHAR := '$0B';
   w_record.XOFFCHAR := '$R';
   w_record.WAITTIME := 2000;
   w_record.MODE := 0;
   w_record.LINE_PRE := 0;
   w_record.BRK_DET := 0;
   w_record.LibSupport := 16#00;
   w_record.res := 16#00;
   r_record.header.block_type := 16#0000;
   r_record.header.block_len := 16#0000;
   r_record.header.block_ver := 16#0000;
   r_record.header.res := 16#0000;
   r_record.SetFtrs := 16#0000;
   r_record.PortCfg := 16#0000;
   r_record.SendCfg := 16#0000;
   r_record.RcvCfg := 16#0000;
   r_record.SgnSet := 16#0000;
   r_record.R3964Err := 16#0000;
END_DATA_BLOCK

DATA_BLOCK "Receive_P2P_DB"   // DB28
// stored: AutoNumber true, DBAccessibleFromOPCUA true, DBAccessibleFromWebserver true, InstanceOfName Receive_P2P, OfSystemLibElement Receive_P2P, OfSystemLibVersion 1.4
"Receive_P2P"
   // VAR_INPUT
   //    PORT : PORT := 306;
   //    BUFFER : Variant;
   // END_VAR
   // VAR_OUTPUT
   //    NDR : Bool := FALSE;
   //    ERROR : Bool := FALSE;
   //    STATUS : Word := 16#7002;
   //    LENGTH : UInt := 0;
   // END_VAR
   // VAR
   //    OldPORT : PORT := 306;
   //    received_length : UInt := 16;
   //    y_ptp_status : SInt := 0;
   //    y_state : SInt := 0;
   //    y_seq_nr : Byte := 16#2E;
   //    safe_h1 : Byte := 16#00;
   //    safe_h2 : Byte := 16#00;
   //    safe_h3 : Byte := 16#00;
   //    safe_h4 : Byte := 16#00;
   //    isClassic : Bool := FALSE;
   //    record_nr : Int := 49;
   //    offset : UDInt := 0;
   //    RDREC { S7_SetPoint := 'True'} : RDREC;
   //    ReceiveBuffer : Array[0..1027] of Byte;
   //    i_addr : UDInt := 6;
   //    mySrcVAREF { ExternalAccessible := 'False'; ExternalVisible := 'False'; ExternalWritable := 'False'; S7_SetPoint := 'True'} : VAREF;
   //    myDstVAREF { ExternalVisible := 'False'; S7_SetPoint := 'True'} : VAREF;
   // END_VAR
BEGIN
   RDREC.REQ := FALSE;
   RDREC.ID := 306;
   RDREC.INDEX := 50;
   RDREC.MLEN := 1028;
   RDREC.VALID := TRUE;
   RDREC.BUSY := FALSE;
   RDREC.ERROR := FALSE;
   RDREC.STATUS := 16#0000_0000;
   RDREC.LEN := 20;
   ReceiveBuffer[0] := 16#2E;
   ReceiveBuffer[1] := 16#01;
   ReceiveBuffer[2] := 16#00;
   ReceiveBuffer[3] := 16#10;
   ReceiveBuffer[4] := 16#30;
   ReceiveBuffer[5] := 16#33;
   ReceiveBuffer[6] := 16#38;
   ReceiveBuffer[7] := 16#30;
   ReceiveBuffer[8] := 16#34;
   ReceiveBuffer[9] := 16#30;
   ReceiveBuffer[10] := 16#37;
   ReceiveBuffer[11] := 16#33;
   ReceiveBuffer[12] := 16#47;
   ReceiveBuffer[13] := 16#4F;
   ReceiveBuffer[14] := 16#32;
   ReceiveBuffer[15] := 16#33;
   ReceiveBuffer[16] := 16#35;
   ReceiveBuffer[17] := 16#34;
   ReceiveBuffer[18] := 16#38;
   ReceiveBuffer[19] := 16#0D;
   ReceiveBuffer[20] := 16#38;
   ReceiveBuffer[21] := 16#35;
   ReceiveBuffer[22] := 16#0D;
   ReceiveBuffer[23..1027] := 16#00;
   mySrcVAREF.RID := 16#0000_0000;
   mySrcVAREF.AREA := 16#00;
   mySrcVAREF.DB_NUMBER := 0;
   mySrcVAREF.OFFSET := 0;
   mySrcVAREF.LENGTH := 0;
   myDstVAREF.RID := 16#0201_0002;
   myDstVAREF.AREA := 16#8B;
   myDstVAREF.DB_NUMBER := 6;
   myDstVAREF.OFFSET := 2184;
   myDstVAREF.LENGTH := 255;
END_DATA_BLOCK

DATA_BLOCK "Receive_Reset_DB2"   // DB39
// stored: AutoNumber true, DBAccessibleFromOPCUA true, DBAccessibleFromWebserver true, InstanceOfName Receive_Reset, OfSystemLibElement Receive_Reset, OfSystemLibVersion 1.2
"Receive_Reset"
   // VAR_INPUT
   //    REQ : Bool := FALSE;
   //    PORT : Word := 16#0132;
   // END_VAR
   // VAR_OUTPUT
   //    DONE : Bool := FALSE;
   //    ERROR : Bool := FALSE;
   //    STATUS : Word := 16#7000;
   // END_VAR
   // VAR
   //    b_e_REQ : Bool := FALSE;
   //    y_state : SInt := 0;
   //    WRREC { S7_SetPoint := 'True'} : WRREC;
   //    w_record { S7_SetPoint := 'True'} : P2P_ResetData;
   // END_VAR
BEGIN
   WRREC.REQ := FALSE;
   WRREC.ID := 306;
   WRREC.INDEX := 54;
   WRREC.LEN := 12;
   WRREC.DONE := TRUE;
   WRREC.BUSY := FALSE;
   WRREC.ERROR := FALSE;
   WRREC.STATUS := 16#0000_0000;
   w_record.header.block_type := 16#0036;
   w_record.header.block_len := 16#0008;
   w_record.header.block_ver := 16#0100;
   w_record.header.res := 16#0000;
   w_record.ackn := 16#01;
   w_record.res1 := 16#00;
   w_record.res2 := 16#00;
   w_record.res3 := 16#00;
END_DATA_BLOCK

DATA_BLOCK "STEP CHANGE TIMER"   // DB11
{ S7_Optimized_Access := 'TRUE' }
// stored: AutoNumber true, DBAccessibleFromOPCUA true, DBAccessibleFromWebserver true, InstanceOfName IEC_TIMER, OfSystemLibElement IEC_TIMER, OfSystemLibVersion 1.0
"IEC_TIMER"
   // VAR
   //    PT : Time := T#500MS;
   //    ET { ExternalWritable := 'False'} : Time;
   //    IN : Bool := FALSE;
   //    Q { ExternalWritable := 'False'} : Bool;
   // END_VAR
BEGIN
END_DATA_BLOCK

DATA_BLOCK "TONR CICLE TIME TIMER"   // DB17
{ S7_Optimized_Access := 'TRUE' }
// stored: AutoNumber true, DBAccessibleFromOPCUA true, DBAccessibleFromWebserver true, InstanceOfName IEC_TIMER, OfSystemLibElement IEC_TIMER, OfSystemLibVersion 1.0
"IEC_TIMER"
   // VAR
   //    PT : Time := T#0MS;
   //    ET { ExternalWritable := 'False'} : Time;
   //    IN : Bool := FALSE;
   //    Q { ExternalWritable := 'False'} : Bool;
   // END_VAR
BEGIN
END_DATA_BLOCK

DATA_BLOCK "TON_Finala_Izq"   // DB12
{ S7_Optimized_Access := 'TRUE' }
// stored: AutoNumber true, DBAccessibleFromOPCUA true, DBAccessibleFromWebserver true, InstanceOfName IEC_TIMER, OfSystemLibElement IEC_TIMER, OfSystemLibVersion 1.0
"IEC_TIMER"
   // VAR
   //    PT : Time := T#0MS;
   //    ET { ExternalWritable := 'False'} : Time;
   //    IN : Bool := FALSE;
   //    Q { ExternalWritable := 'False'} : Bool;
   // END_VAR
BEGIN
END_DATA_BLOCK

DATA_BLOCK "leftTrackProductPokayokeTimer"   // DB30
{ S7_Optimized_Access := 'TRUE' }
// stored: AutoNumber true, DBAccessibleFromOPCUA true, DBAccessibleFromWebserver true, InstanceOfName IEC_TIMER, OfSystemLibElement IEC_TIMER, OfSystemLibVersion 1.0
"IEC_TIMER"
   // VAR
   //    PT : Time := T#500MS;
   //    ET { ExternalWritable := 'False'} : Time;
   //    IN : Bool := FALSE;
   //    Q { ExternalWritable := 'False'} : Bool;
   // END_VAR
BEGIN
END_DATA_BLOCK

DATA_BLOCK "printerFaultTimer"   // DB34
{ S7_Optimized_Access := 'TRUE' }
// stored: AutoNumber true, DBAccessibleFromOPCUA true, DBAccessibleFromWebserver true, InstanceOfName IEC_TIMER, OfSystemLibElement IEC_TIMER, OfSystemLibVersion 1.0
"IEC_TIMER"
   // VAR
   //    PT : Time := T#5S;
   //    ET { ExternalWritable := 'False'} : Time;
   //    IN : Bool := FALSE;
   //    Q { ExternalWritable := 'False'} : Bool;
   // END_VAR
BEGIN
END_DATA_BLOCK

DATA_BLOCK "rightTrackProductPokayokeTimer"   // DB31
{ S7_Optimized_Access := 'TRUE' }
// stored: AutoNumber true, DBAccessibleFromOPCUA true, DBAccessibleFromWebserver true, InstanceOfName IEC_TIMER, OfSystemLibElement IEC_TIMER, OfSystemLibVersion 1.0
"IEC_TIMER"
   // VAR
   //    PT : Time := T#500MS;
   //    ET { ExternalWritable := 'False'} : Time;
   //    IN : Bool := FALSE;
   //    Q { ExternalWritable := 'False'} : Bool;
   // END_VAR
BEGIN
END_DATA_BLOCK

DATA_BLOCK "trigger"   // DB29
{ S7_Optimized_Access := 'TRUE' }
// stored: AutoNumber true, DBAccessibleFromOPCUA true, DBAccessibleFromWebserver true, InstanceOfName IEC_TIMER, OfSystemLibElement IEC_TIMER, OfSystemLibVersion 1.0
"IEC_TIMER"
   // VAR
   //    PT : Time := T#20MS;
   //    ET { ExternalWritable := 'False'} : Time;
   //    IN : Bool := TRUE;
   //    Q { ExternalWritable := 'False'} : Bool;
   // END_VAR
BEGIN
END_DATA_BLOCK

